# B&R Automation Studio project TD52 (part 68)

#### Gen2_ref.h
```c
/********************************************************************
 * COPYRIGHT -- B&R Industrial Automation GmbH
 ********************************************************************
 * Program: Gen2_ref
 * File: Gen2_ref.h
 * Author: 105055527
 * Last modified by: kelleto00
 * Created: Wed Apr 16 13:02:53 2008
 * Last modified: Wed Oct 09 10:01:33 2024
 * Model Version: 4.14.00.04
 * Description: V4.10.00.01, 01-09-2020 Keller, Ke Estimator, additive LS factor, Ptraj SpeedCtrl, LVRT Freeze HLCi
   V4.10.00.01, 02-10-2020 Keller, bugfix HLCi p2srefLX init, BDC_lib: change Inf to 1e7
   V4.10.00.01, 13-11-2020 Keller, bugfix LXcorr T2s/ZZP, LSLff damping, dbgOut for Leanox WG compensation
   V4.10.00.01, 27-01-2021 Keller, Lx WGV compensation: no reset in island mode, addition before skipfire compensation
   V4.10.00.01, 02-02-2021 Keller, initialization lambda estimation with rLam_Start
   V4.11.00.01, 28-05-2021 Keller, Gas Quality Change (GQC) Improvements, LHV estimator output
   V4.11.00.01, 05-11-2021 Keller, Bugfix BDC: worksplit offset, optionally Nset instead of Nnom, rN_Eng_LRskipF
   V4.12.00.01, 10-02-2021 Keller, SpeedCtrl2.0 TU Wien: Disturbance Estimator, LQR incl. droop & leanox
   V4.12.00.02, 23-05-2022 Arnold, Leanox point C in low load
   V4.12.00.02, 09-06-2022 Kafka, add external skip fire input for isolated and grid parallel operation
   V4.12.00.03, 15-09-2022 Keller, add power trajectory to HLCi for extended LQR (Droop setpoint)
   V4.12.00.04, 12-10-2022 Keller, add gas flow comp. factor for rejections
   V4.12.00.05, 13-10-2022 Keller, power filter for static skipfire in island mode
   V4.12.00.06, 15-11-2022 Keller, Ke adaptation with disturbance observer
   V4.13.00.01, 15-11-2022 Keller, FDC: R_mix output, HLCi: R_mix for Ke
   V4.13.00.02, 10-07-2023 Keller, interpolation of LHV, rho_gas and Lmin
   V4.13.00.03, 10-07-2023 Keller, load dependent gas dosage delay
   V4.13.00.04, 11-09-2023 Keller, D-part FSM, bugfix dPTV ramp
   V4.13.00.05, 27-02-2024 Keller, Filter outputs without bSS
   V4.13.00.06, 10-04-2024 Keller, bugfix leanox manual mode with bSepEmisCtrl
   V4.14.00.01, 01-07-2024 Keller, iNskip_LRfor Ke calculation
   V4.14.00.02, 17-09-2024 Keller, Use actual speed for observer disturbance dg (Gen2_ref/HLC_Island (HLC_Island_ref)/iLQR_SF/Ref LQR)
   V4.14.00.03, 30-09-2024 Keller, LR gas flow compensation possible without actuator saturation
   V4.14.00.04, 02-10-2024 Keller, Limit derivative power setpoint for FSM
 * modified Comment:
 ********************************************************************
 * Header for program Gen2_ref
 ********************************************************************
 * Generated with B&R Automation Studio Target for Simulink V6.7.1
 * (ERT based)
 ********************************************************************/

#ifndef RTW_HEADER_Gen2_ref_h_
#define RTW_HEADER_Gen2_ref_h_
#include <math.h>
#ifndef Gen2_ref_COMMON_INCLUDES_
#define Gen2_ref_COMMON_INCLUDES_
#include "rtwtypes.h"
#include "zero_crossing_types.h"
#endif                                 /* Gen2_ref_COMMON_INCLUDES_ */

#include "Gen2_ref_types.h"
#include "lGen2.h"
/* Beginning of Dynamic TypeDefs: */
/* End of Dynamic TypeDefs: */
#ifndef MIN
#define MIN(a,b)	((a) < (b) ? (a) : (b))
#endif

#ifndef MAX
#define MAX(a,b)	((a) > (b) ? (a) : (b))
#endif

#ifndef AST_ROUND
#define AST_ROUND(x) ((x)>=0?(long long)((x)+0.5):(long long)((x)-0.5))
#endif

#include "rt_nonfinite.h"
#include "rt_defines.h"

/* Macros for accessing real-time model data structure */
#ifndef rtmGetBlockIO
#define rtmGetBlockIO(rtm)             ((rtm)->blockIO)
#endif

#ifndef rtmSetBlockIO
#define rtmSetBlockIO(rtm, val)        ((rtm)->blockIO = (val))
#endif

#ifndef rtmGetPrevZCSigState
#define rtmGetPrevZCSigState(rtm)      ((rtm)->prevZCSigState)
#endif

#ifndef rtmSetPrevZCSigState
#define rtmSetPrevZCSigState(rtm, val) ((rtm)->prevZCSigState = (val))
#endif

#ifndef rtmGetRootDWork
#define rtmGetRootDWork(rtm)           ((rtm)->dwork)
#endif

#ifndef rtmSetRootDWork
#define rtmSetRootDWork(rtm, val)      ((rtm)->dwork = (val))
#endif

#ifndef rtmGetY
#define rtmGetY(rtm)                   ((rtm)->outputs)
#endif

#ifndef rtmSetY
#define rtmSetY(rtm, val)              ((rtm)->outputs = (val))
#endif

#ifndef rtmGetErrorStatus
#define rtmGetErrorStatus(rtm)         ((rtm)->errorStatus)
#endif

#ifndef rtmSetErrorStatus
#define rtmSetErrorStatus(rtm, val)    ((rtm)->errorStatus = (val))
#endif

#ifndef MIN
#define MIN(a,b)                       ((a) < (b) ? (a) : (b))
#endif

#ifndef MAX
#define MAX(a,b)                       ((a) > (b) ? (a) : (b))
#endif

#ifndef AST_ROUND
#define AST_ROUND(x)                   ((x)>=0?(long long)((x)+0.5):(long long)((x)-0.5))
#endif

/* Block signals for system '<S23>/Filter1' */

/* Block states (default storage) for system '<S23>/Filter1' */

/* Block signals for system '<S23>/TON_1' */

/* Block states (default storage) for system '<S23>/TON_1' */

/* Block signals for system '<S62>/Filter3' */

/* Block states (default storage) for system '<S62>/Filter3' */

/* Block signals for system '<S24>/MATLAB Function' */

/* Block states (default storage) for system '<S24>/MATLAB Function' */

/* Block signals for system '<S27>/engine massflow' */

/* Block signals for system '<S1>/IntegerZOH' */

/* Block states (default storage) for system '<S1>/IntegerZOH' */

/* Block signals for system '<S144>/lam2cg1' */

/* Block signals for system '<S44>/engine massflow2' */

/* Block signals for system '<S161>/Inverse_Linearization4' */

/* Block signals for system '<S190>/N_TC_HP_filt' */

/* Block states (default storage) for system '<S190>/N_TC_HP_filt' */

/* Block signals for system '<S267>/Mg' */

/* Block signals for system '<S267>/lam2cg1' */

/* Block signals for system '<S305>/FILTER no delay' */

/* Block states (default storage) for system '<S305>/FILTER no delay' */

/* Block signals for system '<S306>/2nd Order Filter' */

/* Block states (default storage) for system '<S306>/2nd Order Filter' */

/* Block signals for system '<S306>/2nd Order Filter3' */

/* Block states (default storage) for system '<S306>/2nd Order Filter3' */

/* Block signals for system '<S6>/TOF' */

/* Block states (default storage) for system '<S6>/TOF' */

/* Block signals for system '<S373>/2-point interpolation, with extrapolation' */

/* Block signals for system '<S379>/MATLAB Function' */

/* Block states (default storage) for system '<S379>/MATLAB Function' */

/* Block signals for system '<S379>/MATLAB Function1' */

/* Block states (default storage) for system '<S379>/MATLAB Function1' */

/* Block signals for system '<S344>/Pd_filt' */

/* Block states (default storage) for system '<S344>/Pd_filt' */

/* Block signals for system '<S426>/TP' */

/* Block states (default storage) for system '<S426>/TP' */

/* Block signals for system '<S427>/TOF' */

/* Block states (default storage) for system '<S427>/TOF' */

/* Block signals for system '<S427>/TP_ActSat_CBV' */

/* Block states (default storage) for system '<S427>/TP_ActSat_CBV' */

/* Block signals for system '<S589>/MATLAB Function' */

/* Block states (default storage) for system '<S589>/MATLAB Function' */

/* Block signals for system '<S630>/Filter' */

/* Block states (default storage) for system '<S630>/Filter' */

/* Block signals for system '<S666>/Ke Map Update' */

/* Block states (default storage) for system '<S666>/Ke Map Update' */

/* Block signals for system '<S666>/MATLAB Function1' */

/* Block states (default storage) for system '<S666>/MATLAB Function1' */

/* Block signals (default storage) */

/* Block states (default storage) for system '<Root>' */

/* Zero-crossing (trigger) state */

/* Invariant block signals for system '<S306>/2nd Order Filter' */

/* Invariant block signals for system '<S306>/2nd Order Filter3' */

/* Invariant block signals for system '<S630>/Filter' */

/* Invariant block signals for system '<S666>/Ke Map Update' */

/* Invariant block signals (default storage) */

/* Constant parameters (default storage) */

/* External outputs (root outports fed by signals with default storage) */

/* Real-time Model Data Structure */

extern const ConstBlockIO_Gen2_ref Gen2_ref_ConstB;/* constant block i/o */

/* Constant parameters (default storage) */
extern const ConstParam_Gen2_ref Gen2_ref_ConstP;

/* Model entry point functions */
extern void Gen2_ref_initialize(RT_MODEL_Gen2_ref *const Gen2_ref_M, struct Gen2* inst);
extern void Gen2_ref_step(RT_MODEL_Gen2_ref *const Gen2_ref_M, struct Gen2* inst);
extern void Gen2_ref_terminate(RT_MODEL_Gen2_ref *const Gen2_ref_M, struct Gen2* inst);

/*-
 * The generated code includes comments that allow you to trace directly
 * back to the appropriate location in the model.  The basic format
 * is <system>/block_name, where system is the system number (uniquely
 * assigned by Simulink) and block_name is the name of the block.
 *
 * Use the MATLAB hilite_system command to trace the generated code back
 * to the model.  For example,
 *
 * hilite_system('<S3>')    - opens system 3
 * hilite_system('<S3>/Kp') - opens and selects block Kp which resides in S3
 *
 * Here is the system hierarchy for this model
 *
 * '<Root>' : 'Gen2_ref'
 * '<S1>'   : 'Gen2_ref/BDC'
 * '<S2>'   : 'Gen2_ref/DocBlock'
 * '<S3>'   : 'Gen2_ref/EFF'
 * '<S4>'   : 'Gen2_ref/EngineSignals'
 * '<S5>'   : 'Gen2_ref/FDC'
 * '<S6>'   : 'Gen2_ref/Gas Quality Change'
 * '<S7>'   : 'Gen2_ref/HLC_Grid'
 * '<S8>'   : 'Gen2_ref/HLC_Island'
 * '<S9>'   : 'Gen2_ref/ITC'
 * '<S10>'  : 'Gen2_ref/Info'
 * '<S11>'  : 'Gen2_ref/Interpolation gas 1//2&3 specific parameters'
 * '<S12>'  : 'Gen2_ref/Ke Estimator NetP'
 * '<S13>'  : 'Gen2_ref/LHV estimator'
 * '<S14>'  : 'Gen2_ref/LambdaLimit'
 * '<S15>'  : 'Gen2_ref/Leanox_Comp_WG'
 * '<S16>'  : 'Gen2_ref/Outputs'
 * '<S17>'  : 'Gen2_ref/Power trajectory'
 * '<S18>'  : 'Gen2_ref/Saturation Det'
 * '<S19>'  : 'Gen2_ref/Skipfire'
 * '<S20>'  : 'Gen2_ref/SteadyState'
 * '<S21>'  : 'Gen2_ref/brake eff estimate'
 * '<S22>'  : 'Gen2_ref/BDC/ TC Protection'
 * '<S23>'  : 'Gen2_ref/BDC/1_Motion_Planning3'
 * '<S24>'  : 'Gen2_ref/BDC/2_Approach_selector_TV'
 * '<S25>'  : 'Gen2_ref/BDC/Approach_selector_CBV'
 * '<S26>'  : 'Gen2_ref/BDC/CBV_Control'
 * '<S27>'  : 'Gen2_ref/BDC/CBV_Feedforward'
 * '<S28>'  : 'Gen2_ref/BDC/Compare To Constant'
 * '<S29>'  : 'Gen2_ref/BDC/Compare To Constant1'
 * '<S30>'  : 'Gen2_ref/BDC/Compare To Constant2'
 * '<S31>'  : 'Gen2_ref/BDC/Difference1'
 * '<S32>'  : 'Gen2_ref/BDC/Divisor'
 * '<S33>'  : 'Gen2_ref/BDC/Divisor1'
 * '<S34>'  : 'Gen2_ref/BDC/Divisor2'
 * '<S35>'  : 'Gen2_ref/BDC/Divisor3'
 * '<S36>'  : 'Gen2_ref/BDC/DocBlock'
 * '<S37>'  : 'Gen2_ref/BDC/IntegerZOH'
 * '<S38>'  : 'Gen2_ref/BDC/IntegerZOH1'
 * '<S39>'  : 'Gen2_ref/BDC/IntegerZOH2'
 * '<S40>'  : 'Gen2_ref/BDC/Model Info'
 * '<S41>'  : 'Gen2_ref/BDC/PID_para'
 * '<S42>'  : 'Gen2_ref/BDC/Saturation Dynamic'
 * '<S43>'  : 'Gen2_ref/BDC/SurgeProtection'
 * '<S44>'  : 'Gen2_ref/BDC/TV_Feedforward'
 * '<S45>'  : 'Gen2_ref/BDC/Throttle_Control'
 * '<S46>'  : 'Gen2_ref/BDC/WGV_Feedforward'
 * '<S47>'  : 'Gen2_ref/BDC/ TC Protection/Compare To Zero'
 * '<S48>'  : 'Gen2_ref/BDC/1_Motion_Planning3/Delta_ref'
 * '<S49>'  : 'Gen2_ref/BDC/1_Motion_Planning3/Filter1'
 * '<S50>'  : 'Gen2_ref/BDC/1_Motion_Planning3/Filter2'
 * '<S51>'  : 'Gen2_ref/BDC/1_Motion_Planning3/Filter4'
 * '<S52>'  : 'Gen2_ref/BDC/1_Motion_Planning3/Rate Limit'
 * '<S53>'  : 'Gen2_ref/BDC/1_Motion_Planning3/Reset_'
 * '<S54>'  : 'Gen2_ref/BDC/1_Motion_Planning3/Saturation Dynamic'
 * '<S55>'  : 'Gen2_ref/BDC/1_Motion_Planning3/Saturation Dynamic1'
 * '<S56>'  : 'Gen2_ref/BDC/1_Motion_Planning3/Saturation Dynamic2'
 * '<S57>'  : 'Gen2_ref/BDC/1_Motion_Planning3/Saturation Dynamic3'
 * '<S58>'  : 'Gen2_ref/BDC/1_Motion_Planning3/Saturation Dynamic4'
 * '<S59>'  : 'Gen2_ref/BDC/1_Motion_Planning3/Saturation Dynamic5'
 * '<S60>'  : 'Gen2_ref/BDC/1_Motion_Planning3/Saturation Dynamic6'
 * '<S61>'  : 'Gen2_ref/BDC/1_Motion_Planning3/TON_1'
 * '<S62>'  : 'Gen2_ref/BDC/1_Motion_Planning3/offset for LEANOX tracking if TV open'
 * '<S63>'  : 'Gen2_ref/BDC/1_Motion_Planning3/rateLimit'
 * '<S64>'  : 'Gen2_ref/BDC/1_Motion_Planning3/rateLimit1'
 * '<S65>'  : 'Gen2_ref/BDC/1_Motion_Planning3/ref traj'
 * '<S66>'  : 'Gen2_ref/BDC/1_Motion_Planning3/Delta_ref/Compare To Zero'
 * '<S67>'  : 'Gen2_ref/BDC/1_Motion_Planning3/Delta_ref/Divisor'
 * '<S68>'  : 'Gen2_ref/BDC/1_Motion_Planning3/Delta_ref/Divisor1'
 * '<S69>'  : 'Gen2_ref/BDC/1_Motion_Planning3/Delta_ref/Divisor/Data Type Conversion Inherited'
 * '<S70>'  : 'Gen2_ref/BDC/1_Motion_Planning3/Delta_ref/Divisor1/Data Type Conversion Inherited'
 * '<S71>'  : 'Gen2_ref/BDC/1_Motion_Planning3/Filter1/Divisor'
 * '<S72>'  : 'Gen2_ref/BDC/1_Motion_Planning3/Filter1/Divisor/Data Type Conversion Inherited'
 * '<S73>'  : 'Gen2_ref/BDC/1_Motion_Planning3/Filter2/Divisor'
 * '<S74>'  : 'Gen2_ref/BDC/1_Motion_Planning3/Filter2/Divisor/Data Type Conversion Inherited'
 * '<S75>'  : 'Gen2_ref/BDC/1_Motion_Planning3/Filter4/Divisor'
 * '<S76>'  : 'Gen2_ref/BDC/1_Motion_Planning3/Filter4/Divisor/Data Type Conversion Inherited'
 * '<S77>'  : 'Gen2_ref/BDC/1_Motion_Planning3/Rate Limit/slewratelimit_rejection CBV'
 * '<S78>'  : 'Gen2_ref/BDC/1_Motion_Planning3/Rate Limit/slewratelimit_rejection TV'
 * '<S79>'  : 'Gen2_ref/BDC/1_Motion_Planning3/Rate Limit/slewratelimit_rejection CBV/rateLimit'
 * '<S80>'  : 'Gen2_ref/BDC/1_Motion_Planning3/Rate Limit/slewratelimit_rejection CBV/rateLimit1'
 * '<S81>'  : 'Gen2_ref/BDC/1_Motion_Planning3/Rate Limit/slewratelimit_rejection CBV/rateLimit2'
 * '<S82>'  : 'Gen2_ref/BDC/1_Motion_Planning3/Rate Limit/slewratelimit_rejection CBV/rateLimit3'
 * '<S83>'  : 'Gen2_ref/BDC/1_Motion_Planning3/Rate Limit/slewratelimit_rejection CBV/rateLimit/Saturation Dynamic'
 * '<S84>'  : 'Gen2_ref/BDC/1_Motion_Planning3/Rate Limit/slewratelimit_rejection CBV/rateLimit1/Saturation Dynamic'
 * '<S85>'  : 'Gen2_ref/BDC/1_Motion_Planning3/Rate Limit/slewratelimit_rejection CBV/rateLimit2/Saturation Dynamic'
 * '<S86>'  : 'Gen2_ref/BDC/1_Motion_Planning3/Rate Limit/slewratelimit_rejection CBV/rateLimit3/Saturation Dynamic'
 * '<S87>'  : 'Gen2_ref/BDC/1_Motion_Planning3/Rate Limit/slewratelimit_rejection TV/rateLimit'
 * '<S88>'  : 'Gen2_ref/BDC/1_Motion_Planning3/Rate Limit/slewratelimit_rejection TV/rateLimit1'
 * '<S89>'  : 'Gen2_ref/BDC/1_Motion_Planning3/Rate Limit/slewratelimit_rejection TV/rateLimit2'
 * '<S90>'  : 'Gen2_ref/BDC/1_Motion_Planning3/Rate Limit/slewratelimit_rejection TV/rateLimit3'
 * '<S91>'  : 'Gen2_ref/BDC/1_Motion_Planning3/Rate Limit/slewratelimit_rejection TV/rateLimit/Saturation Dynamic'
 * '<S92>'  : 'Gen2_ref/BDC/1_Motion_Planning3/Rate Limit/slewratelimit_rejection TV/rateLimit1/Saturation Dynamic'
 * '<S93>'  : 'Gen2_ref/BDC/1_Motion_Planning3/Rate Limit/slewratelimit_rejection TV/rateLimit2/Saturation Dynamic'
 * '<S94>'  : 'Gen2_ref/BDC/1_Motion_Planning3/Rate Limit/slewratelimit_rejection TV/rateLimit3/Saturation Dynamic'
 * '<S95>'  : 'Gen2_ref/BDC/1_Motion_Planning3/TON_1/Data Type Conversion Inherited'
 * '<S96>'  : 'Gen2_ref/BDC/1_Motion_Planning3/offset for LEANOX tracking if TV open/Divisor'
 * '<S97>'  : 'Gen2_ref/BDC/1_Motion_Planning3/offset for LEANOX tracking if TV open/Filter3'
 * '<S98>'  : 'Gen2_ref/BDC/1_Motion_Planning3/offset for LEANOX tracking if TV open/MATLAB Function'
 * '<S99>'  : 'Gen2_ref/BDC/1_Motion_Planning3/offset for LEANOX tracking if TV open/Divisor/Data Type Conversion Inherited'
 * '<S100>' : 'Gen2_ref/BDC/1_Motion_Planning3/offset for LEANOX tracking if TV open/Filter3/Divisor'
 * '<S101>' : 'Gen2_ref/BDC/1_Motion_Planning3/offset for LEANOX tracking if TV open/Filter3/Divisor/Data Type Conversion Inherited'
 * '<S102>' : 'Gen2_ref/BDC/1_Motion_Planning3/rateLimit/Saturation Dynamic'
 * '<S103>' : 'Gen2_ref/BDC/1_Motion_Planning3/rateLimit1/Saturation Dynamic'
 * '<S104>' : 'Gen2_ref/BDC/2_Approach_selector_TV/MATLAB Function'
 * '<S105>' : 'Gen2_ref/BDC/Approach_selector_CBV/MATLAB Function'
 * '<S106>' : 'Gen2_ref/BDC/Approach_selector_CBV/Saturation Dynamic'
 * '<S107>' : 'Gen2_ref/BDC/CBV_Control/Detect Change'
 * '<S108>' : 'Gen2_ref/BDC/CBV_Control/Saturation Dynamic'
 * '<S109>' : 'Gen2_ref/BDC/CBV_Control/Saturation Dynamic1'
 * '<S110>' : 'Gen2_ref/BDC/CBV_Control/fb_err'
 * '<S111>' : 'Gen2_ref/BDC/CBV_Control/reset init'
 * '<S112>' : 'Gen2_ref/BDC/CBV_Feedforward/Divisor'
 * '<S113>' : 'Gen2_ref/BDC/CBV_Feedforward/MATLAB Function1'
 * '<S114>' : 'Gen2_ref/BDC/CBV_Feedforward/Saturation Dynamic'
 * '<S115>' : 'Gen2_ref/BDC/CBV_Feedforward/Saturation Dynamic1'
 * '<S116>' : 'Gen2_ref/BDC/CBV_Feedforward/cbv tracking1'
 * '<S117>' : 'Gen2_ref/BDC/CBV_Feedforward/dynamic_massflow '
 * '<S118>' : 'Gen2_ref/BDC/CBV_Feedforward/engine massflow'
 * '<S119>' : 'Gen2_ref/BDC/CBV_Feedforward/engine massflow1'
 * '<S120>' : 'Gen2_ref/BDC/CBV_Feedforward/Divisor/Data Type Conversion Inherited'
 * '<S121>' : 'Gen2_ref/BDC/CBV_Feedforward/cbv tracking1/Compare To Constant'
 * '<S122>' : 'Gen2_ref/BDC/CBV_Feedforward/cbv tracking1/Compare To Constant1'
 * '<S123>' : 'Gen2_ref/BDC/CBV_Feedforward/cbv tracking1/Saturation Dynamic'
 * '<S124>' : 'Gen2_ref/BDC/Divisor/Data Type Conversion Inherited'
 * '<S125>' : 'Gen2_ref/BDC/Divisor1/Data Type Conversion Inherited'
 * '<S126>' : 'Gen2_ref/BDC/Divisor2/Data Type Conversion Inherited'
 * '<S127>' : 'Gen2_ref/BDC/Divisor3/Data Type Conversion Inherited'
 * '<S128>' : 'Gen2_ref/BDC/PID_para/Saturation Dynamic'
 * '<S129>' : 'Gen2_ref/BDC/PID_para/Saturation Dynamic1'
 * '<S130>' : 'Gen2_ref/BDC/PID_para/Saturation Dynamic2'
 * '<S131>' : 'Gen2_ref/BDC/PID_para/Saturation Dynamic3'
 * '<S132>' : 'Gen2_ref/BDC/PID_para/p2s fitler2'
 * '<S133>' : 'Gen2_ref/BDC/SurgeProtection/SP'
 * '<S134>' : 'Gen2_ref/BDC/SurgeProtection/SP2'
 * '<S135>' : 'Gen2_ref/BDC/SurgeProtection/SP/Divisor'
 * '<S136>' : 'Gen2_ref/BDC/SurgeProtection/SP/Saturation Dynamic'
 * '<S137>' : 'Gen2_ref/BDC/SurgeProtection/SP/Saturation Dynamic1'
 * '<S138>' : 'Gen2_ref/BDC/SurgeProtection/SP/Divisor/Data Type Conversion Inherited'
 * '<S139>' : 'Gen2_ref/BDC/SurgeProtection/SP2/Divisor'
 * '<S140>' : 'Gen2_ref/BDC/SurgeProtection/SP2/Divisor2'
 * '<S141>' : 'Gen2_ref/BDC/SurgeProtection/SP2/Filter'
 * '<S142>' : 'Gen2_ref/BDC/SurgeProtection/SP2/MATLAB Function'
 * '<S143>' : 'Gen2_ref/BDC/SurgeProtection/SP2/MATLAB Function1'
 * '<S144>' : 'Gen2_ref/BDC/SurgeProtection/SP2/MassFlowCalc'
 * '<S145>' : 'Gen2_ref/BDC/SurgeProtection/SP2/Divisor/Data Type Conversion Inherited'
 * '<S146>' : 'Gen2_ref/BDC/SurgeProtection/SP2/Divisor2/Data Type Conversion Inherited'
 * '<S147>' : 'Gen2_ref/BDC/SurgeProtection/SP2/Filter/Divisor'
 * '<S148>' : 'Gen2_ref/BDC/SurgeProtection/SP2/Filter/Divisor/Data Type Conversion Inherited'
 * '<S149>' : 'Gen2_ref/BDC/SurgeProtection/SP2/MassFlowCalc/Divisor2'
 * '<S150>' : 'Gen2_ref/BDC/SurgeProtection/SP2/MassFlowCalc/lam2cg1'
 * '<S151>' : 'Gen2_ref/BDC/SurgeProtection/SP2/MassFlowCalc/Divisor2/Data Type Conversion Inherited'
 * '<S152>' : 'Gen2_ref/BDC/SurgeProtection/SP2/MassFlowCalc/lam2cg1/Divisor'
 * '<S153>' : 'Gen2_ref/BDC/SurgeProtection/SP2/MassFlowCalc/lam2cg1/Divisor/Data Type Conversion Inherited'
 * '<S154>' : 'Gen2_ref/BDC/TV_Feedforward/Divisor'
 * '<S155>' : 'Gen2_ref/BDC/TV_Feedforward/Dyn_Term'
 * '<S156>' : 'Gen2_ref/BDC/TV_Feedforward/MATLAB Function3'
 * '<S157>' : 'Gen2_ref/BDC/TV_Feedforward/Saturation Dynamic1'
 * '<S158>' : 'Gen2_ref/BDC/TV_Feedforward/engine massflow2'
 * '<S159>' : 'Gen2_ref/BDC/TV_Feedforward/Divisor/Data Type Conversion Inherited'
 * '<S160>' : 'Gen2_ref/BDC/Throttle_Control/Detect Change'
 * '<S161>' : 'Gen2_ref/BDC/Throttle_Control/Integrator Init'
 * '<S162>' : 'Gen2_ref/BDC/Throttle_Control/Inverse_Linearization1'
 * '<S163>' : 'Gen2_ref/BDC/Throttle_Control/Inverse_Linearization2'
 * '<S164>' : 'Gen2_ref/BDC/Throttle_Control/Inverse_Linearization3'
 * '<S165>' : 'Gen2_ref/BDC/Throttle_Control/Inverse_Linearization4'
 * '<S166>' : 'Gen2_ref/BDC/Throttle_Control/Linearization'
 * '<S167>' : 'Gen2_ref/BDC/Throttle_Control/Saturation Dynamic'
 * '<S168>' : 'Gen2_ref/BDC/Throttle_Control/tv_fb_err'
 * '<S169>' : 'Gen2_ref/BDC/Throttle_Control/Integrator Init/Inverse_Linearization4'
 * '<S170>' : 'Gen2_ref/BDC/WGV_Feedforward/Divisor'
 * '<S171>' : 'Gen2_ref/BDC/WGV_Feedforward/MATLAB Function1'
 * '<S172>' : 'Gen2_ref/BDC/WGV_Feedforward/Saturation Dynamic'
 * '<S173>' : 'Gen2_ref/BDC/WGV_Feedforward/Saturation Dynamic1'
 * '<S174>' : 'Gen2_ref/BDC/WGV_Feedforward/cbv tracking1'
 * '<S175>' : 'Gen2_ref/BDC/WGV_Feedforward/dynamic_massflow'
 * '<S176>' : 'Gen2_ref/BDC/WGV_Feedforward/engine massflow'
 * '<S177>' : 'Gen2_ref/BDC/WGV_Feedforward/engine massflow1'
 * '<S178>' : 'Gen2_ref/BDC/WGV_Feedforward/Divisor/Data Type Conversion Inherited'
 * '<S179>' : 'Gen2_ref/BDC/WGV_Feedforward/cbv tracking1/Compare To Constant'
 * '<S180>' : 'Gen2_ref/BDC/WGV_Feedforward/cbv tracking1/Saturation Dynamic'
 * '<S181>' : 'Gen2_ref/BDC/WGV_Feedforward/cbv tracking1/TP'
 * '<S182>' : 'Gen2_ref/BDC/WGV_Feedforward/cbv tracking1/TP/Compare To Zero'
 * '<S183>' : 'Gen2_ref/BDC/WGV_Feedforward/cbv tracking1/TP/Enabled Subsystem'
 * '<S184>' : 'Gen2_ref/BDC/WGV_Feedforward/cbv tracking1/TP/Enabled Subsystem1'
 * '<S185>' : 'Gen2_ref/BDC/WGV_Feedforward/cbv tracking1/TP/Rate Limiter'
 * '<S186>' : 'Gen2_ref/BDC/WGV_Feedforward/cbv tracking1/TP/Rate Limiter/Saturation Dynamic'
 * '<S187>' : 'Gen2_ref/EngineSignals/Compare To Constant'
 * '<S188>' : 'Gen2_ref/EngineSignals/Compare To Constant1'
 * '<S189>' : 'Gen2_ref/EngineSignals/Compare To Constant3'
 * '<S190>' : 'Gen2_ref/EngineSignals/IgnAvg'
 * '<S191>' : 'Gen2_ref/EngineSignals/N_TC_HP_filt'
 * '<S192>' : 'Gen2_ref/EngineSignals/N_TC_LP_filt'
 * '<S193>' : 'Gen2_ref/EngineSignals/N_TC_LP_filt1'
 * '<S194>' : 'Gen2_ref/EngineSignals/Pel_filt'
 * '<S195>' : 'Gen2_ref/EngineSignals/T1HP_filt'
 * '<S196>' : 'Gen2_ref/EngineSignals/T1LP_filt'
 * '<S197>' : 'Gen2_ref/EngineSignals/T2s_filt'
 * '<S198>' : 'Gen2_ref/EngineSignals/T3HP_filt'
 * '<S199>' : 'Gen2_ref/EngineSignals/T3LP_filt'
 * '<S200>' : 'Gen2_ref/EngineSignals/T4LP_filt'
 * '<S201>' : 'Gen2_ref/EngineSignals/Volt_filt'
 * '<S202>' : 'Gen2_ref/EngineSignals/p1HP_filt'
 * '<S203>' : 'Gen2_ref/EngineSignals/p1LP_filt'
 * '<S204>' : 'Gen2_ref/EngineSignals/p2HP_filt'
 * '<S205>' : 'Gen2_ref/EngineSignals/p2s_filt'
 * '<S206>' : 'Gen2_ref/EngineSignals/p3LP_filt'
 * '<S207>' : 'Gen2_ref/EngineSignals/p3LP_filt1'
 * '<S208>' : 'Gen2_ref/EngineSignals/p4LP_filt'
 * '<S209>' : 'Gen2_ref/EngineSignals/IgnAvg/N_TC_HP_filt'
 * '<S210>' : 'Gen2_ref/EngineSignals/IgnAvg/N_TC_HP_filt/Divisor'
 * '<S211>' : 'Gen2_ref/EngineSignals/IgnAvg/N_TC_HP_filt/Divisor/Data Type Conversion Inherited'
 * '<S212>' : 'Gen2_ref/EngineSignals/N_TC_HP_filt/N_TC_HP_filt'
 * '<S213>' : 'Gen2_ref/EngineSignals/N_TC_HP_filt/N_TC_HP_filt/Divisor'
 * '<S214>' : 'Gen2_ref/EngineSignals/N_TC_HP_filt/N_TC_HP_filt/Divisor/Data Type Conversion Inherited'
 * '<S215>' : 'Gen2_ref/EngineSignals/N_TC_LP_filt/N_TC_LP_filt'
 * '<S216>' : 'Gen2_ref/EngineSignals/N_TC_LP_filt/N_TC_LP_filt/Divisor'
 * '<S217>' : 'Gen2_ref/EngineSignals/N_TC_LP_filt/N_TC_LP_filt/Divisor/Data Type Conversion Inherited'
 * '<S218>' : 'Gen2_ref/EngineSignals/N_TC_LP_filt1/N_TC_LP_filt'
 * '<S219>' : 'Gen2_ref/EngineSignals/N_TC_LP_filt1/N_TC_LP_filt/Divisor'
 * '<S220>' : 'Gen2_ref/EngineSignals/N_TC_LP_filt1/N_TC_LP_filt/Divisor/Data Type Conversion Inherited'
 * '<S221>' : 'Gen2_ref/EngineSignals/Pel_filt/Pel_filt'
 * '<S222>' : 'Gen2_ref/EngineSignals/Pel_filt/Pel_filt/Divisor'
 * '<S223>' : 'Gen2_ref/EngineSignals/Pel_filt/Pel_filt/Divisor/Data Type Conversion Inherited'
 * '<S224>' : 'Gen2_ref/EngineSignals/T1HP_filt/T1HP_filt'
 * '<S225>' : 'Gen2_ref/EngineSignals/T1HP_filt/T1HP_filt/Divisor'
 * '<S226>' : 'Gen2_ref/EngineSignals/T1HP_filt/T1HP_filt/Divisor/Data Type Conversion Inherited'
 * '<S227>' : 'Gen2_ref/EngineSignals/T1LP_filt/T1LP_filt'
 * '<S228>' : 'Gen2_ref/EngineSignals/T1LP_filt/T1LP_filt/Divisor'
 * '<S229>' : 'Gen2_ref/EngineSignals/T1LP_filt/T1LP_filt/Divisor/Data Type Conversion Inherited'
 * '<S230>' : 'Gen2_ref/EngineSignals/T2s_filt/T2s_filt'
 * '<S231>' : 'Gen2_ref/EngineSignals/T2s_filt/T2s_filt/Divisor'
 * '<S232>' : 'Gen2_ref/EngineSignals/T2s_filt/T2s_filt/Divisor/Data Type Conversion Inherited'
 * '<S233>' : 'Gen2_ref/EngineSignals/T3HP_filt/T3HP_filt'
 * '<S234>' : 'Gen2_ref/EngineSignals/T3HP_filt/T3HP_filt/Divisor'
 * '<S235>' : 'Gen2_ref/EngineSignals/T3HP_filt/T3HP_filt/Divisor/Data Type Conversion Inherited'
 * '<S236>' : 'Gen2_ref/EngineSignals/T3LP_filt/T3LP_filt'
 * '<S237>' : 'Gen2_ref/EngineSignals/T3LP_filt/T3LP_filt/Divisor'
 * '<S238>' : 'Gen2_ref/EngineSignals/T3LP_filt/T3LP_filt/Divisor/Data Type Conversion Inherited'
 * '<S239>' : 'Gen2_ref/EngineSignals/T4LP_filt/T3LP_filt'
 * '<S240>' : 'Gen2_ref/EngineSignals/T4LP_filt/T3LP_filt/Divisor'
 * '<S241>' : 'Gen2_ref/EngineSignals/T4LP_filt/T3LP_filt/Divisor/Data Type Conversion Inherited'
 * '<S242>' : 'Gen2_ref/EngineSignals/Volt_filt/Volt_filt'
 * '<S243>' : 'Gen2_ref/EngineSignals/Volt_filt/Volt_filt/Divisor'
 * '<S244>' : 'Gen2_ref/EngineSignals/Volt_filt/Volt_filt/Divisor/Data Type Conversion Inherited'
 * '<S245>' : 'Gen2_ref/EngineSignals/p1HP_filt/p1HP_filt'
 * '<S246>' : 'Gen2_ref/EngineSignals/p1HP_filt/p1HP_filt/Divisor'
 * '<S247>' : 'Gen2_ref/EngineSignals/p1HP_filt/p1HP_filt/Divisor/Data Type Conversion Inherited'
 * '<S248>' : 'Gen2_ref/EngineSignals/p1LP_filt/Filter'
 * '<S249>' : 'Gen2_ref/EngineSignals/p1LP_filt/Filter/Divisor'
 * '<S250>' : 'Gen2_ref/EngineSignals/p1LP_filt/Filter/Divisor/Data Type Conversion Inherited'
 * '<S251>' : 'Gen2_ref/EngineSignals/p2HP_filt/p2HP_filt'
 * '<S252>' : 'Gen2_ref/EngineSignals/p2HP_filt/p2HP_filt/Divisor'
 * '<S253>' : 'Gen2_ref/EngineSignals/p2HP_filt/p2HP_filt/Divisor/Data Type Conversion Inherited'
 * '<S254>' : 'Gen2_ref/EngineSignals/p2s_filt/p2s_filt'
 * '<S255>' : 'Gen2_ref/EngineSignals/p2s_filt/p2s_filt/Divisor'
 * '<S256>' : 'Gen2_ref/EngineSignals/p2s_filt/p2s_filt/Divisor/Data Type Conversion Inherited'
 * '<S257>' : 'Gen2_ref/EngineSignals/p3LP_filt/p3LP_filt'
 * '<S258>' : 'Gen2_ref/EngineSignals/p3LP_filt/p3LP_filt/Divisor'
 * '<S259>' : 'Gen2_ref/EngineSignals/p3LP_filt/p3LP_filt/Divisor/Data Type Conversion Inherited'
 * '<S260>' : 'Gen2_ref/EngineSignals/p3LP_filt1/p3LP_filt'
 * '<S261>' : 'Gen2_ref/EngineSignals/p3LP_filt1/p3LP_filt/Divisor'
 * '<S262>' : 'Gen2_ref/EngineSignals/p3LP_filt1/p3LP_filt/Divisor/Data Type Conversion Inherited'
 * '<S263>' : 'Gen2_ref/EngineSignals/p4LP_filt/p4LP_filt'
 * '<S264>' : 'Gen2_ref/EngineSignals/p4LP_filt/p4LP_filt/Divisor'
 * '<S265>' : 'Gen2_ref/EngineSignals/p4LP_filt/p4LP_filt/Divisor/Data Type Conversion Inherited'
 * '<S266>' : 'Gen2_ref/FDC/DocBlock'
 * '<S267>' : 'Gen2_ref/FDC/GasArt12'
 * '<S268>' : 'Gen2_ref/FDC/GasArt3'
 * '<S269>' : 'Gen2_ref/FDC/IntegerZOH'
 * '<S270>' : 'Gen2_ref/FDC/IntegerZOH1'
 * '<S271>' : 'Gen2_ref/FDC/Model Info'
 * '<S272>' : 'Gen2_ref/FDC/Signal Conditioning'
 * '<S273>' : 'Gen2_ref/FDC/GasArt12/Divisor'
 * '<S274>' : 'Gen2_ref/FDC/GasArt12/Mg'
 * '<S275>' : 'Gen2_ref/FDC/GasArt12/Safety check logic'
 * '<S276>' : 'Gen2_ref/FDC/GasArt12/lam2cg'
 * '<S277>' : 'Gen2_ref/FDC/GasArt12/lam2cg1'
 * '<S278>' : 'Gen2_ref/FDC/GasArt12/Divisor/Data Type Conversion Inherited'
 * '<S279>' : 'Gen2_ref/FDC/GasArt12/Mg/Divisor'
 * '<S280>' : 'Gen2_ref/FDC/GasArt12/Mg/Divisor/Data Type Conversion Inherited'
 * '<S281>' : 'Gen2_ref/FDC/GasArt12/Safety check logic/Divisor1'
 * '<S282>' : 'Gen2_ref/FDC/GasArt12/Safety check logic/Divisor2'
 * '<S283>' : 'Gen2_ref/FDC/GasArt12/Safety check logic/Divisor1/Data Type Conversion Inherited'
 * '<S284>' : 'Gen2_ref/FDC/GasArt12/Safety check logic/Divisor2/Data Type Conversion Inherited'
 * '<S285>' : 'Gen2_ref/FDC/GasArt12/lam2cg/Divisor'
 * '<S286>' : 'Gen2_ref/FDC/GasArt12/lam2cg/Divisor/Data Type Conversion Inherited'
 * '<S287>' : 'Gen2_ref/FDC/GasArt12/lam2cg1/Divisor'
 * '<S288>' : 'Gen2_ref/FDC/GasArt12/lam2cg1/Divisor/Data Type Conversion Inherited'
 * '<S289>' : 'Gen2_ref/FDC/GasArt3/Divisor'
 * '<S290>' : 'Gen2_ref/FDC/GasArt3/Mg'
 * '<S291>' : 'Gen2_ref/FDC/GasArt3/Safety check logic'
 * '<S292>' : 'Gen2_ref/FDC/GasArt3/lam2cg'
 * '<S293>' : 'Gen2_ref/FDC/GasArt3/lam2cg1'
 * '<S294>' : 'Gen2_ref/FDC/GasArt3/Divisor/Data Type Conversion Inherited'
 * '<S295>' : 'Gen2_ref/FDC/GasArt3/Mg/Divisor'
 * '<S296>' : 'Gen2_ref/FDC/GasArt3/Mg/Divisor/Data Type Conversion Inherited'
 * '<S297>' : 'Gen2_ref/FDC/GasArt3/Safety check logic/Divisor1'
 * '<S298>' : 'Gen2_ref/FDC/GasArt3/Safety check logic/Divisor2'
 * '<S299>' : 'Gen2_ref/FDC/GasArt3/Safety check logic/Divisor1/Data Type Conversion Inherited'
 * '<S300>' : 'Gen2_ref/FDC/GasArt3/Safety check logic/Divisor2/Data Type Conversion Inherited'
 * '<S301>' : 'Gen2_ref/FDC/GasArt3/lam2cg/Divisor'
 * '<S302>' : 'Gen2_ref/FDC/GasArt3/lam2cg/Divisor/Data Type Conversion Inherited'
 * '<S303>' : 'Gen2_ref/FDC/GasArt3/lam2cg1/Divisor'
 * '<S304>' : 'Gen2_ref/FDC/GasArt3/lam2cg1/Divisor/Data Type Conversion Inherited'
 * '<S305>' : 'Gen2_ref/FDC/Signal Conditioning/first order filter'
 * '<S306>' : 'Gen2_ref/FDC/Signal Conditioning/second order filter'
 * '<S307>' : 'Gen2_ref/FDC/Signal Conditioning/transient switching'
 * '<S308>' : 'Gen2_ref/FDC/Signal Conditioning/first order filter/FILTER no delay'
 * '<S309>' : 'Gen2_ref/FDC/Signal Conditioning/first order filter/FILTER no delay1'
 * '<S310>' : 'Gen2_ref/FDC/Signal Conditioning/first order filter/FILTER no delay2'
 * '<S311>' : 'Gen2_ref/FDC/Signal Conditioning/first order filter/FILTER no delay3'
 * '<S312>' : 'Gen2_ref/FDC/Signal Conditioning/first order filter/FILTER no delay4'
 * '<S313>' : 'Gen2_ref/FDC/Signal Conditioning/first order filter/FILTER no delay5'
 * '<S314>' : 'Gen2_ref/FDC/Signal Conditioning/second order filter/2nd Order Filter'
 * '<S315>' : 'Gen2_ref/FDC/Signal Conditioning/second order filter/2nd Order Filter1'
 * '<S316>' : 'Gen2_ref/FDC/Signal Conditioning/second order filter/2nd Order Filter2'
 * '<S317>' : 'Gen2_ref/FDC/Signal Conditioning/second order filter/2nd Order Filter3'
 * '<S318>' : 'Gen2_ref/FDC/Signal Conditioning/second order filter/2nd Order Filter4'
 * '<S319>' : 'Gen2_ref/FDC/Signal Conditioning/second order filter/2nd Order Filter/Divisor1'
 * '<S320>' : 'Gen2_ref/FDC/Signal Conditioning/second order filter/2nd Order Filter/Divisor1/Data Type Conversion Inherited'
 * '<S321>' : 'Gen2_ref/FDC/Signal Conditioning/second order filter/2nd Order Filter1/Divisor1'
 * '<S322>' : 'Gen2_ref/FDC/Signal Conditioning/second order filter/2nd Order Filter1/Divisor1/Data Type Conversion Inherited'
 * '<S323>' : 'Gen2_ref/FDC/Signal Conditioning/second order filter/2nd Order Filter2/Divisor1'
 * '<S324>' : 'Gen2_ref/FDC/Signal Conditioning/second order filter/2nd Order Filter2/Divisor1/Data Type Conversion Inherited'
 * '<S325>' : 'Gen2_ref/FDC/Signal Conditioning/second order filter/2nd Order Filter3/Divisor1'
 * '<S326>' : 'Gen2_ref/FDC/Signal Conditioning/second order filter/2nd Order Filter3/Divisor1/Data Type Conversion Inherited'
 * '<S327>' : 'Gen2_ref/FDC/Signal Conditioning/second order filter/2nd Order Filter4/Divisor1'
 * '<S328>' : 'Gen2_ref/FDC/Signal Conditioning/second order filter/2nd Order Filter4/Divisor1/Data Type Conversion Inherited'
 * '<S329>' : 'Gen2_ref/Gas Quality Change/TOF'
 * '<S330>' : 'Gen2_ref/Gas Quality Change/TOF1'
 * '<S331>' : 'Gen2_ref/Gas Quality Change/TOF2'
 * '<S332>' : 'Gen2_ref/Gas Quality Change/TON'
 * '<S333>' : 'Gen2_ref/Gas Quality Change/TOF/Data Type Conversion Inherited'
 * '<S334>' : 'Gen2_ref/Gas Quality Change/TOF1/Data Type Conversion Inherited'
 * '<S335>' : 'Gen2_ref/Gas Quality Change/TOF2/Data Type Conversion Inherited'
 * '<S336>' : 'Gen2_ref/Gas Quality Change/TON/Data Type Conversion Inherited'
 * '<S337>' : 'Gen2_ref/HLC_Grid/DocBlock'
 * '<S338>' : 'Gen2_ref/HLC_Grid/LEANOX map'
 * '<S339>' : 'Gen2_ref/HLC_Grid/LVRT_React'
 * '<S340>' : 'Gen2_ref/HLC_Grid/MBC_FF'
 * '<S341>' : 'Gen2_ref/HLC_Grid/Model Info'
 * '<S342>' : 'Gen2_ref/HLC_Grid/Power_Ctrl'
 * '<S343>' : 'Gen2_ref/HLC_Grid/Power_Ctrl Gas Quality Change'
 * '<S344>' : 'Gen2_ref/HLC_Grid/Power_Trajectory'
 * '<S345>' : 'Gen2_ref/HLC_Grid/Subsystem Reference'
 * '<S346>' : 'Gen2_ref/HLC_Grid/LEANOX map/Divisor'
 * '<S347>' : 'Gen2_ref/HLC_Grid/LEANOX map/Divisor1'
 * '<S348>' : 'Gen2_ref/HLC_Grid/LEANOX map/Divisor10'
 * '<S349>' : 'Gen2_ref/HLC_Grid/LEANOX map/Divisor11'
 * '<S350>' : 'Gen2_ref/HLC_Grid/LEANOX map/Divisor12'
 * '<S351>' : 'Gen2_ref/HLC_Grid/LEANOX map/Divisor2'
 * '<S352>' : 'Gen2_ref/HLC_Grid/LEANOX map/Divisor3'
 * '<S353>' : 'Gen2_ref/HLC_Grid/LEANOX map/Divisor4'
 * '<S354>' : 'Gen2_ref/HLC_Grid/LEANOX map/Divisor5'
 * '<S355>' : 'Gen2_ref/HLC_Grid/LEANOX map/Divisor6'
 * '<S356>' : 'Gen2_ref/HLC_Grid/LEANOX map/Divisor7'
 * '<S357>' : 'Gen2_ref/HLC_Grid/LEANOX map/Divisor8'
 * '<S358>' : 'Gen2_ref/HLC_Grid/LEANOX map/Divisor9'
 * '<S359>' : 'Gen2_ref/HLC_Grid/LEANOX map/LeanoxCorr'
 * '<S360>' : 'Gen2_ref/HLC_Grid/LEANOX map/Divisor/Data Type Conversion Inherited'
 * '<S361>' : 'Gen2_ref/HLC_Grid/LEANOX map/Divisor1/Data Type Conversion Inherited'
 * '<S362>' : 'Gen2_ref/HLC_Grid/LEANOX map/Divisor10/Data Type Conversion Inherited'
 * '<S363>' : 'Gen2_ref/HLC_Grid/LEANOX map/Divisor11/Data Type Conversion Inherited'
 * '<S364>' : 'Gen2_ref/HLC_Grid/LEANOX map/Divisor12/Data Type Conversion Inherited'
 * '<S365>' : 'Gen2_ref/HLC_Grid/LEANOX map/Divisor2/Data Type Conversion Inherited'
 * '<S366>' : 'Gen2_ref/HLC_Grid/LEANOX map/Divisor3/Data Type Conversion Inherited'
 * '<S367>' : 'Gen2_ref/HLC_Grid/LEANOX map/Divisor4/Data Type Conversion Inherited'
 * '<S368>' : 'Gen2_ref/HLC_Grid/LEANOX map/Divisor5/Data Type Conversion Inherited'
 * '<S369>' : 'Gen2_ref/HLC_Grid/LEANOX map/Divisor6/Data Type Conversion Inherited'
 * '<S370>' : 'Gen2_ref/HLC_Grid/LEANOX map/Divisor7/Data Type Conversion Inherited'
 * '<S371>' : 'Gen2_ref/HLC_Grid/LEANOX map/Divisor8/Data Type Conversion Inherited'
 * '<S372>' : 'Gen2_ref/HLC_Grid/LEANOX map/Divisor9/Data Type Conversion Inherited'
 * '<S373>' : 'Gen2_ref/HLC_Grid/LEANOX map/LeanoxCorr/Leanox_Comp'
 * '<S374>' : 'Gen2_ref/HLC_Grid/LEANOX map/LeanoxCorr/Leanox_Comp/2-point interpolation, with extrapolation'
 * '<S375>' : 'Gen2_ref/HLC_Grid/LEANOX map/LeanoxCorr/Leanox_Comp/2-point interpolation, with extrapolation1'
 * '<S376>' : 'Gen2_ref/HLC_Grid/LEANOX map/LeanoxCorr/Leanox_Comp/Saturation Dynamic'
 * '<S377>' : 'Gen2_ref/HLC_Grid/LEANOX map/LeanoxCorr/Leanox_Comp/Saturation Dynamic1'
 * '<S378>' : 'Gen2_ref/HLC_Grid/LVRT_React/MATLAB Function'
 * '<S379>' : 'Gen2_ref/HLC_Grid/Power_Ctrl/PID_Power'
 * '<S380>' : 'Gen2_ref/HLC_Grid/Power_Ctrl/Saturation Dynamic7'
 * '<S381>' : 'Gen2_ref/HLC_Grid/Power_Ctrl/Texh_limit'
 * '<S382>' : 'Gen2_ref/HLC_Grid/Power_Ctrl/PID_Power/MATLAB Function'
 * '<S383>' : 'Gen2_ref/HLC_Grid/Power_Ctrl/PID_Power/MATLAB Function1'
 * '<S384>' : 'Gen2_ref/HLC_Grid/Power_Ctrl/PID_Power/Saturation Dynamic'
 * '<S385>' : 'Gen2_ref/HLC_Grid/Power_Ctrl/PID_Power/rateLimit'
 * '<S386>' : 'Gen2_ref/HLC_Grid/Power_Ctrl/PID_Power/rateLimit/Saturation Dynamic'
 * '<S387>' : 'Gen2_ref/HLC_Grid/Power_Ctrl/Texh_limit/Saturation Dynamic4'
 * '<S388>' : 'Gen2_ref/HLC_Grid/Power_Ctrl Gas Quality Change/Anti Wind Up'
 * '<S389>' : 'Gen2_ref/HLC_Grid/Power_Ctrl Gas Quality Change/PID_Power'
 * '<S390>' : 'Gen2_ref/HLC_Grid/Power_Ctrl Gas Quality Change/Anti Wind Up/Saturation Dynamic'
 * '<S391>' : 'Gen2_ref/HLC_Grid/Power_Ctrl Gas Quality Change/PID_Power/MATLAB Function'
 * '<S392>' : 'Gen2_ref/HLC_Grid/Power_Ctrl Gas Quality Change/PID_Power/MATLAB Function1'
 * '<S393>' : 'Gen2_ref/HLC_Grid/Power_Ctrl Gas Quality Change/PID_Power/Saturation Dynamic'
 * '<S394>' : 'Gen2_ref/HLC_Grid/Power_Ctrl Gas Quality Change/PID_Power/rateLimit'
 * '<S395>' : 'Gen2_ref/HLC_Grid/Power_Ctrl Gas Quality Change/PID_Power/rateLimit/Saturation Dynamic'
 * '<S396>' : 'Gen2_ref/HLC_Grid/Power_Trajectory/Pd_filt'
 * '<S397>' : 'Gen2_ref/HLC_Grid/Power_Trajectory/Saturation Dynamic'
 * '<S398>' : 'Gen2_ref/HLC_Grid/Power_Trajectory/Saturation Dynamic1'
 * '<S399>' : 'Gen2_ref/HLC_Grid/Power_Trajectory/Saturation Dynamic2'
 * '<S400>' : 'Gen2_ref/HLC_Grid/Power_Trajectory/Saturation Dynamic3'
 * '<S401>' : 'Gen2_ref/HLC_Grid/Power_Trajectory/Saturation Dynamic4'
 * '<S402>' : 'Gen2_ref/HLC_Grid/Power_Trajectory/WO1'
 * '<S403>' : 'Gen2_ref/HLC_Grid/Power_Trajectory/WO2'
 * '<S404>' : 'Gen2_ref/HLC_Grid/Power_Trajectory/rateLimit'
 * '<S405>' : 'Gen2_ref/HLC_Grid/Power_Trajectory/Pd_filt/Divisor'
 * '<S406>' : 'Gen2_ref/HLC_Grid/Power_Trajectory/Pd_filt/Divisor/Data Type Conversion Inherited'
 * '<S407>' : 'Gen2_ref/HLC_Grid/Power_Trajectory/WO1/Divisor'
 * '<S408>' : 'Gen2_ref/HLC_Grid/Power_Trajectory/WO1/Divisor/Data Type Conversion Inherited'
 * '<S409>' : 'Gen2_ref/HLC_Grid/Power_Trajectory/WO2/Divisor'
 * '<S410>' : 'Gen2_ref/HLC_Grid/Power_Trajectory/WO2/Divisor/Data Type Conversion Inherited'
 * '<S411>' : 'Gen2_ref/HLC_Grid/Power_Trajectory/rateLimit/Saturation Dynamic'
 * '<S412>' : 'Gen2_ref/HLC_Grid/Subsystem Reference/p2sfilt'
 * '<S413>' : 'Gen2_ref/HLC_Grid/Subsystem Reference/rateLimit1'
 * '<S414>' : 'Gen2_ref/HLC_Grid/Subsystem Reference/p2sfilt/Divisor'
 * '<S415>' : 'Gen2_ref/HLC_Grid/Subsystem Reference/p2sfilt/Divisor/Data Type Conversion Inherited'
 * '<S416>' : 'Gen2_ref/HLC_Grid/Subsystem Reference/rateLimit1/Saturation Dynamic'
 * '<S417>' : 'Gen2_ref/HLC_Island/BDC_Trajectory'
 * '<S418>' : 'Gen2_ref/HLC_Island/CalcPowerRot'
 * '<S419>' : 'Gen2_ref/HLC_Island/DocBlock'
 * '<S420>' : 'Gen2_ref/HLC_Island/Filter'
 * '<S421>' : 'Gen2_ref/HLC_Island/IntegerZOH'
 * '<S422>' : 'Gen2_ref/HLC_Island/LEANOX ERR Correction Transient'
 * '<S423>' : 'Gen2_ref/HLC_Island/LEANOX map'
 * '<S424>' : 'Gen2_ref/HLC_Island/LSL Interface'
 * '<S425>' : 'Gen2_ref/HLC_Island/LVRT freeze'
 * '<S426>' : 'Gen2_ref/HLC_Island/Load Rejection transient compensation'
 * '<S427>' : 'Gen2_ref/HLC_Island/LoadRejection'
 * '<S428>' : 'Gen2_ref/HLC_Island/Model Info'
 * '<S429>' : 'Gen2_ref/HLC_Island/Skip_control'
 * '<S430>' : 'Gen2_ref/HLC_Island/Subsystem'
 * '<S431>' : 'Gen2_ref/HLC_Island/iLQR_SF'
 * '<S432>' : 'Gen2_ref/HLC_Island/p2sFF'
 * '<S433>' : 'Gen2_ref/HLC_Island/BDC_Trajectory/p2sfilt'
 * '<S434>' : 'Gen2_ref/HLC_Island/BDC_Trajectory/rateLimit1'
 * '<S435>' : 'Gen2_ref/HLC_Island/BDC_Trajectory/p2sfilt/Divisor'
 * '<S436>' : 'Gen2_ref/HLC_Island/BDC_Trajectory/p2sfilt/Divisor/Data Type Conversion Inherited'
 * '<S437>' : 'Gen2_ref/HLC_Island/BDC_Trajectory/rateLimit1/Saturation Dynamic'
 * '<S438>' : 'Gen2_ref/HLC_Island/CalcPowerRot/2nd Order Filter'
 * '<S439>' : 'Gen2_ref/HLC_Island/CalcPowerRot/Filter'
 * '<S440>' : 'Gen2_ref/HLC_Island/CalcPowerRot/2nd Order Filter/Divisor1'
 * '<S441>' : 'Gen2_ref/HLC_Island/CalcPowerRot/2nd Order Filter/Divisor1/Data Type Conversion Inherited'
 * '<S442>' : 'Gen2_ref/HLC_Island/CalcPowerRot/Filter/Divisor'
 * '<S443>' : 'Gen2_ref/HLC_Island/CalcPowerRot/Filter/Divisor/Data Type Conversion Inherited'
 * '<S444>' : 'Gen2_ref/HLC_Island/Filter/Divisor'
 * '<S445>' : 'Gen2_ref/HLC_Island/Filter/Divisor/Data Type Conversion Inherited'
 * '<S446>' : 'Gen2_ref/HLC_Island/LEANOX map/Divisor'
 * '<S447>' : 'Gen2_ref/HLC_Island/LEANOX map/Divisor1'
 * '<S448>' : 'Gen2_ref/HLC_Island/LEANOX map/Divisor10'
 * '<S449>' : 'Gen2_ref/HLC_Island/LEANOX map/Divisor11'
 * '<S450>' : 'Gen2_ref/HLC_Island/LEANOX map/Divisor12'
 * '<S451>' : 'Gen2_ref/HLC_Island/LEANOX map/Divisor2'
 * '<S452>' : 'Gen2_ref/HLC_Island/LEANOX map/Divisor3'
 * '<S453>' : 'Gen2_ref/HLC_Island/LEANOX map/Divisor4'
 * '<S454>' : 'Gen2_ref/HLC_Island/LEANOX map/Divisor5'
 * '<S455>' : 'Gen2_ref/HLC_Island/LEANOX map/Divisor6'
 * '<S456>' : 'Gen2_ref/HLC_Island/LEANOX map/Divisor7'
 * '<S457>' : 'Gen2_ref/HLC_Island/LEANOX map/Divisor8'
 * '<S458>' : 'Gen2_ref/HLC_Island/LEANOX map/Divisor9'
 * '<S459>' : 'Gen2_ref/HLC_Island/LEANOX map/LeanoxCorr'
 * '<S460>' : 'Gen2_ref/HLC_Island/LEANOX map/Divisor/Data Type Conversion Inherited'
 * '<S461>' : 'Gen2_ref/HLC_Island/LEANOX map/Divisor1/Data Type Conversion Inherited'
 * '<S462>' : 'Gen2_ref/HLC_Island/LEANOX map/Divisor10/Data Type Conversion Inherited'
 * '<S463>' : 'Gen2_ref/HLC_Island/LEANOX map/Divisor11/Data Type Conversion Inherited'
 * '<S464>' : 'Gen2_ref/HLC_Island/LEANOX map/Divisor12/Data Type Conversion Inherited'
 * '<S465>' : 'Gen2_ref/HLC_Island/LEANOX map/Divisor2/Data Type Conversion Inherited'
 * '<S466>' : 'Gen2_ref/HLC_Island/LEANOX map/Divisor3/Data Type Conversion Inherited'
 * '<S467>' : 'Gen2_ref/HLC_Island/LEANOX map/Divisor4/Data Type Conversion Inherited'
 * '<S468>' : 'Gen2_ref/HLC_Island/LEANOX map/Divisor5/Data Type Conversion Inherited'
 * '<S469>' : 'Gen2_ref/HLC_Island/LEANOX map/Divisor6/Data Type Conversion Inherited'
 * '<S470>' : 'Gen2_ref/HLC_Island/LEANOX map/Divisor7/Data Type Conversion Inherited'
 * '<S471>' : 'Gen2_ref/HLC_Island/LEANOX map/Divisor8/Data Type Conversion Inherited'
 * '<S472>' : 'Gen2_ref/HLC_Island/LEANOX map/Divisor9/Data Type Conversion Inherited'
 * '<S473>' : 'Gen2_ref/HLC_Island/LEANOX map/LeanoxCorr/Leanox_Comp'
 * '<S474>' : 'Gen2_ref/HLC_Island/LEANOX map/LeanoxCorr/Leanox_Comp/2-point interpolation, with extrapolation'
 * '<S475>' : 'Gen2_ref/HLC_Island/LEANOX map/LeanoxCorr/Leanox_Comp/2-point interpolation, with extrapolation1'
 * '<S476>' : 'Gen2_ref/HLC_Island/LEANOX map/LeanoxCorr/Leanox_Comp/Saturation Dynamic'
 * '<S477>' : 'Gen2_ref/HLC_Island/LEANOX map/LeanoxCorr/Leanox_Comp/Saturation Dynamic1'
 * '<S478>' : 'Gen2_ref/HLC_Island/LSL Interface/Filter1'
 * '<S479>' : 'Gen2_ref/HLC_Island/LSL Interface/Saturation Dynamic'
 * '<S480>' : 'Gen2_ref/HLC_Island/LSL Interface/speed Filter'
 * '<S481>' : 'Gen2_ref/HLC_Island/LSL Interface/Filter1/Divisor'
 * '<S482>' : 'Gen2_ref/HLC_Island/LSL Interface/Filter1/Divisor/Data Type Conversion Inherited'
 * '<S483>' : 'Gen2_ref/HLC_Island/LSL Interface/speed Filter/Divisor'
 * '<S484>' : 'Gen2_ref/HLC_Island/LSL Interface/speed Filter/Divisor/Data Type Conversion Inherited'
 * '<S485>' : 'Gen2_ref/HLC_Island/LVRT freeze/Filter'
 * '<S486>' : 'Gen2_ref/HLC_Island/LVRT freeze/TOF'
 * '<S487>' : 'Gen2_ref/HLC_Island/LVRT freeze/Filter/Divisor'
 * '<S488>' : 'Gen2_ref/HLC_Island/LVRT freeze/Filter/Divisor/Data Type Conversion Inherited'
 * '<S489>' : 'Gen2_ref/HLC_Island/LVRT freeze/TOF/Data Type Conversion Inherited'
 * '<S490>' : 'Gen2_ref/HLC_Island/Load Rejection transient compensation/Detect Saturation at LR'
 * '<S491>' : 'Gen2_ref/HLC_Island/Load Rejection transient compensation/Hysterese'
 * '<S492>' : 'Gen2_ref/HLC_Island/Load Rejection transient compensation/TP'
 * '<S493>' : 'Gen2_ref/HLC_Island/Load Rejection transient compensation/TP1'
 * '<S494>' : 'Gen2_ref/HLC_Island/Load Rejection transient compensation/rateLimit'
 * '<S495>' : 'Gen2_ref/HLC_Island/Load Rejection transient compensation/TP/Compare To Zero'
 * '<S496>' : 'Gen2_ref/HLC_Island/Load Rejection transient compensation/TP/Enabled Subsystem'
 * '<S497>' : 'Gen2_ref/HLC_Island/Load Rejection transient compensation/TP/Enabled Subsystem1'
 * '<S498>' : 'Gen2_ref/HLC_Island/Load Rejection transient compensation/TP/Rate Limiter'
 * '<S499>' : 'Gen2_ref/HLC_Island/Load Rejection transient compensation/TP/Rate Limiter/Saturation Dynamic'
 * '<S500>' : 'Gen2_ref/HLC_Island/Load Rejection transient compensation/TP1/Compare To Zero'
 * '<S501>' : 'Gen2_ref/HLC_Island/Load Rejection transient compensation/TP1/Enabled Subsystem'
 * '<S502>' : 'Gen2_ref/HLC_Island/Load Rejection transient compensation/TP1/Enabled Subsystem1'
 * '<S503>' : 'Gen2_ref/HLC_Island/Load Rejection transient compensation/TP1/Rate Limiter'
 * '<S504>' : 'Gen2_ref/HLC_Island/Load Rejection transient compensation/TP1/Rate Limiter/Saturation Dynamic'
 * '<S505>' : 'Gen2_ref/HLC_Island/Load Rejection transient compensation/rateLimit/Saturation Dynamic'
 * '<S506>' : 'Gen2_ref/HLC_Island/LoadRejection/Divisor'
 * '<S507>' : 'Gen2_ref/HLC_Island/LoadRejection/Divisor1'
 * '<S508>' : 'Gen2_ref/HLC_Island/LoadRejection/Divisor2'
 * '<S509>' : 'Gen2_ref/HLC_Island/LoadRejection/Divisor3'
 * '<S510>' : 'Gen2_ref/HLC_Island/LoadRejection/Saturation Dynamic'
 * '<S511>' : 'Gen2_ref/HLC_Island/LoadRejection/TOF'
 * '<S512>' : 'Gen2_ref/HLC_Island/LoadRejection/TOF1'
 * '<S513>' : 'Gen2_ref/HLC_Island/LoadRejection/TOF2'
 * '<S514>' : 'Gen2_ref/HLC_Island/LoadRejection/TOF3'
 * '<S515>' : 'Gen2_ref/HLC_Island/LoadRejection/TP'
 * '<S516>' : 'Gen2_ref/HLC_Island/LoadRejection/TP_ActSat_CBV'
 * '<S517>' : 'Gen2_ref/HLC_Island/LoadRejection/TP_ActSat_TV'
 * '<S518>' : 'Gen2_ref/HLC_Island/LoadRejection/TP_Ign retard'
 * '<S519>' : 'Gen2_ref/HLC_Island/LoadRejection/TP_Misfire_OFF'
 * '<S520>' : 'Gen2_ref/HLC_Island/LoadRejection/TP_Misfire_OFF1'
 * '<S521>' : 'Gen2_ref/HLC_Island/LoadRejection/TP_Misfire_OFF2'
 * '<S522>' : 'Gen2_ref/HLC_Island/LoadRejection/TP_Misfire_ON'
 * '<S523>' : 'Gen2_ref/HLC_Island/LoadRejection/TP_Misfire_ON_2nd time'
 * '<S524>' : 'Gen2_ref/HLC_Island/LoadRejection/rateLimit'
 * '<S525>' : 'Gen2_ref/HLC_Island/LoadRejection/Divisor/Data Type Conversion Inherited'
 * '<S526>' : 'Gen2_ref/HLC_Island/LoadRejection/Divisor1/Data Type Conversion Inherited'
 * '<S527>' : 'Gen2_ref/HLC_Island/LoadRejection/Divisor2/Data Type Conversion Inherited'
 * '<S528>' : 'Gen2_ref/HLC_Island/LoadRejection/Divisor3/Data Type Conversion Inherited'
 * '<S529>' : 'Gen2_ref/HLC_Island/LoadRejection/TOF/Data Type Conversion Inherited'
 * '<S530>' : 'Gen2_ref/HLC_Island/LoadRejection/TOF1/Data Type Conversion Inherited'
 * '<S531>' : 'Gen2_ref/HLC_Island/LoadRejection/TOF2/Data Type Conversion Inherited'
 * '<S532>' : 'Gen2_ref/HLC_Island/LoadRejection/TOF3/Data Type Conversion Inherited'
 * '<S533>' : 'Gen2_ref/HLC_Island/LoadRejection/TP/Compare To Zero'
 * '<S534>' : 'Gen2_ref/HLC_Island/LoadRejection/TP/Enabled Subsystem'
 * '<S535>' : 'Gen2_ref/HLC_Island/LoadRejection/TP/Enabled Subsystem1'
 * '<S536>' : 'Gen2_ref/HLC_Island/LoadRejection/TP/Rate Limiter'
 * '<S537>' : 'Gen2_ref/HLC_Island/LoadRejection/TP/Rate Limiter/Saturation Dynamic'
 * '<S538>' : 'Gen2_ref/HLC_Island/LoadRejection/TP_ActSat_CBV/Compare To Zero'
 * '<S539>' : 'Gen2_ref/HLC_Island/LoadRejection/TP_ActSat_CBV/Enabled Subsystem'
 * '<S540>' : 'Gen2_ref/HLC_Island/LoadRejection/TP_ActSat_CBV/Enabled Subsystem1'
 * '<S541>' : 'Gen2_ref/HLC_Island/LoadRejection/TP_ActSat_CBV/Rate Limiter'
 * '<S542>' : 'Gen2_ref/HLC_Island/LoadRejection/TP_ActSat_CBV/Rate Limiter/Saturation Dynamic'
 * '<S543>' : 'Gen2_ref/HLC_Island/LoadRejection/TP_ActSat_TV/Compare To Zero'
 * '<S544>' : 'Gen2_ref/HLC_Island/LoadRejection/TP_ActSat_TV/Enabled Subsystem'
 * '<S545>' : 'Gen2_ref/HLC_Island/LoadRejection/TP_ActSat_TV/Enabled Subsystem1'
 * '<S546>' : 'Gen2_ref/HLC_Island/LoadRejection/TP_ActSat_TV/Rate Limiter'
 * '<S547>' : 'Gen2_ref/HLC_Island/LoadRejection/TP_ActSat_TV/Rate Limiter/Saturation Dynamic'
 * '<S548>' : 'Gen2_ref/HLC_Island/LoadRejection/TP_Ign retard/Compare To Zero'
 * '<S549>' : 'Gen2_ref/HLC_Island/LoadRejection/TP_Ign retard/Enabled Subsystem'
 * '<S550>' : 'Gen2_ref/HLC_Island/LoadRejection/TP_Ign retard/Enabled Subsystem1'
 * '<S551>' : 'Gen2_ref/HLC_Island/LoadRejection/TP_Ign retard/Rate Limiter'
 * '<S552>' : 'Gen2_ref/HLC_Island/LoadRejection/TP_Ign retard/Rate Limiter/Saturation Dynamic'
 * '<S553>' : 'Gen2_ref/HLC_Island/LoadRejection/TP_Misfire_OFF/Compare To Zero'
 * '<S554>' : 'Gen2_ref/HLC_Island/LoadRejection/TP_Misfire_OFF/Enabled Subsystem'
 * '<S555>' : 'Gen2_ref/HLC_Island/LoadRejection/TP_Misfire_OFF/Enabled Subsystem1'
 * '<S556>' : 'Gen2_ref/HLC_Island/LoadRejection/TP_Misfire_OFF/Rate Limiter'
 * '<S557>' : 'Gen2_ref/HLC_Island/LoadRejection/TP_Misfire_OFF/Rate Limiter/Saturation Dynamic'
 * '<S558>' : 'Gen2_ref/HLC_Island/LoadRejection/TP_Misfire_OFF1/Compare To Zero'
 * '<S559>' : 'Gen2_ref/HLC_Island/LoadRejection/TP_Misfire_OFF1/Enabled Subsystem'
 * '<S560>' : 'Gen2_ref/HLC_Island/LoadRejection/TP_Misfire_OFF1/Enabled Subsystem1'
 * '<S561>' : 'Gen2_ref/HLC_Island/LoadRejection/TP_Misfire_OFF1/Rate Limiter'
 * '<S562>' : 'Gen2_ref/HLC_Island/LoadRejection/TP_Misfire_OFF1/Rate Limiter/Saturation Dynamic'
 * '<S563>' : 'Gen2_ref/HLC_Island/LoadRejection/TP_Misfire_OFF2/Compare To Zero'
 * '<S564>' : 'Gen2_ref/HLC_Island/LoadRejection/TP_Misfire_OFF2/Enabled Subsystem'
 * '<S565>' : 'Gen2_ref/HLC_Island/LoadRejection/TP_Misfire_OFF2/Enabled Subsystem1'
 * '<S566>' : 'Gen2_ref/HLC_Island/LoadRejection/TP_Misfire_OFF2/Rate Limiter'
 * '<S567>' : 'Gen2_ref/HLC_Island/LoadRejection/TP_Misfire_OFF2/Rate Limiter/Saturation Dynamic'
 * '<S568>' : 'Gen2_ref/HLC_Island/LoadRejection/TP_Misfire_ON/Compare To Zero'
 * '<S569>' : 'Gen2_ref/HLC_Island/LoadRejection/TP_Misfire_ON/Enabled Subsystem'
 * '<S570>' : 'Gen2_ref/HLC_Island/LoadRejection/TP_Misfire_ON/Enabled Subsystem1'
 * '<S571>' : 'Gen2_ref/HLC_Island/LoadRejection/TP_Misfire_ON/Rate Limiter'
 * '<S572>' : 'Gen2_ref/HLC_Island/LoadRejection/TP_Misfire_ON/Rate Limiter/Saturation Dynamic'
 * '<S573>' : 'Gen2_ref/HLC_Island/LoadRejection/TP_Misfire_ON_2nd time/Compare To Zero'
 * '<S574>' : 'Gen2_ref/HLC_Island/LoadRejection/TP_Misfire_ON_2nd time/Enabled Subsystem'
 * '<S575>' : 'Gen2_ref/HLC_Island/LoadRejection/TP_Misfire_ON_2nd time/Enabled Subsystem1'
 * '<S576>' : 'Gen2_ref/HLC_Island/LoadRejection/TP_Misfire_ON_2nd time/Rate Limiter'
 * '<S577>' : 'Gen2_ref/HLC_Island/LoadRejection/TP_Misfire_ON_2nd time/Rate Limiter/Saturation Dynamic'
 * '<S578>' : 'Gen2_ref/HLC_Island/LoadRejection/rateLimit/Saturation Dynamic'
 * '<S579>' : 'Gen2_ref/HLC_Island/Skip_control/Filter lam lambda_map_adaption1'
 * '<S580>' : 'Gen2_ref/HLC_Island/Skip_control/Lookup Skipfire'
 * '<S581>' : 'Gen2_ref/HLC_Island/Skip_control/pulsed_skipfire_LR'
 * '<S582>' : 'Gen2_ref/HLC_Island/Skip_control/skipfire_LR_notPulsed'
 * '<S583>' : 'Gen2_ref/HLC_Island/Skip_control/Filter lam lambda_map_adaption1/Divisor'
 * '<S584>' : 'Gen2_ref/HLC_Island/Skip_control/Filter lam lambda_map_adaption1/Divisor/Data Type Conversion Inherited'
 * '<S585>' : 'Gen2_ref/HLC_Island/Skip_control/Lookup Skipfire/Lookup Skipfire Static'
 * '<S586>' : 'Gen2_ref/HLC_Island/Skip_control/Lookup Skipfire/lambda control'
 * '<S587>' : 'Gen2_ref/HLC_Island/Skip_control/Lookup Skipfire/Lookup Skipfire Static/Filter'
 * '<S588>' : 'Gen2_ref/HLC_Island/Skip_control/Lookup Skipfire/Lookup Skipfire Static/Filter1'
 * '<S589>' : 'Gen2_ref/HLC_Island/Skip_control/Lookup Skipfire/Lookup Skipfire Static/Look  up Skipfire'
 * '<S590>' : 'Gen2_ref/HLC_Island/Skip_control/Lookup Skipfire/Lookup Skipfire Static/Saturation Dynamic'
 * '<S591>' : 'Gen2_ref/HLC_Island/Skip_control/Lookup Skipfire/Lookup Skipfire Static/Saturation Dynamic1'
 * '<S592>' : 'Gen2_ref/HLC_Island/Skip_control/Lookup Skipfire/Lookup Skipfire Static/Filter/Divisor'
 * '<S593>' : 'Gen2_ref/HLC_Island/Skip_control/Lookup Skipfire/Lookup Skipfire Static/Filter/Divisor/Data Type Conversion Inherited'
 * '<S594>' : 'Gen2_ref/HLC_Island/Skip_control/Lookup Skipfire/Lookup Skipfire Static/Filter1/Divisor'
 * '<S595>' : 'Gen2_ref/HLC_Island/Skip_control/Lookup Skipfire/Lookup Skipfire Static/Filter1/Divisor/Data Type Conversion Inherited'
 * '<S596>' : 'Gen2_ref/HLC_Island/Skip_control/Lookup Skipfire/Lookup Skipfire Static/Look  up Skipfire/Divisor'
 * '<S597>' : 'Gen2_ref/HLC_Island/Skip_control/Lookup Skipfire/Lookup Skipfire Static/Look  up Skipfire/MATLAB Function'
 * '<S598>' : 'Gen2_ref/HLC_Island/Skip_control/Lookup Skipfire/Lookup Skipfire Static/Look  up Skipfire/Saturation Dynamic'
 * '<S599>' : 'Gen2_ref/HLC_Island/Skip_control/Lookup Skipfire/Lookup Skipfire Static/Look  up Skipfire/Divisor/Data Type Conversion Inherited'
 * '<S600>' : 'Gen2_ref/HLC_Island/Skip_control/Lookup Skipfire/lambda control/Divisor'
 * '<S601>' : 'Gen2_ref/HLC_Island/Skip_control/Lookup Skipfire/lambda control/MATLAB Function'
 * '<S602>' : 'Gen2_ref/HLC_Island/Skip_control/Lookup Skipfire/lambda control/Divisor/Data Type Conversion Inherited'
 * '<S603>' : 'Gen2_ref/HLC_Island/Skip_control/pulsed_skipfire_LR/Detect Increase'
 * '<S604>' : 'Gen2_ref/HLC_Island/Skip_control/pulsed_skipfire_LR/Divisor'
 * '<S605>' : 'Gen2_ref/HLC_Island/Skip_control/pulsed_skipfire_LR/Divisor2'
 * '<S606>' : 'Gen2_ref/HLC_Island/Skip_control/pulsed_skipfire_LR/Hysteresis1'
 * '<S607>' : 'Gen2_ref/HLC_Island/Skip_control/pulsed_skipfire_LR/Saturation Dynamic'
 * '<S608>' : 'Gen2_ref/HLC_Island/Skip_control/pulsed_skipfire_LR/pulsewidth modulation'
 * '<S609>' : 'Gen2_ref/HLC_Island/Skip_control/pulsed_skipfire_LR/Divisor/Data Type Conversion Inherited'
 * '<S610>' : 'Gen2_ref/HLC_Island/Skip_control/pulsed_skipfire_LR/Divisor2/Data Type Conversion Inherited'
 * '<S611>' : 'Gen2_ref/HLC_Island/Skip_control/pulsed_skipfire_LR/pulsewidth modulation/Detect Decrease'
 * '<S612>' : 'Gen2_ref/HLC_Island/Skip_control/pulsed_skipfire_LR/pulsewidth modulation/Divisor'
 * '<S613>' : 'Gen2_ref/HLC_Island/Skip_control/pulsed_skipfire_LR/pulsewidth modulation/SkipPulseWaitTP'
 * '<S614>' : 'Gen2_ref/HLC_Island/Skip_control/pulsed_skipfire_LR/pulsewidth modulation/Divisor/Data Type Conversion Inherited'
 * '<S615>' : 'Gen2_ref/HLC_Island/Skip_control/pulsed_skipfire_LR/pulsewidth modulation/SkipPulseWaitTP/Compare To Zero'
 * '<S616>' : 'Gen2_ref/HLC_Island/Skip_control/pulsed_skipfire_LR/pulsewidth modulation/SkipPulseWaitTP/Enabled Subsystem'
 * '<S617>' : 'Gen2_ref/HLC_Island/Skip_control/pulsed_skipfire_LR/pulsewidth modulation/SkipPulseWaitTP/Enabled Subsystem1'
 * '<S618>' : 'Gen2_ref/HLC_Island/Skip_control/pulsed_skipfire_LR/pulsewidth modulation/SkipPulseWaitTP/Rate Limiter'
 * '<S619>' : 'Gen2_ref/HLC_Island/Skip_control/pulsed_skipfire_LR/pulsewidth modulation/SkipPulseWaitTP/Rate Limiter/Saturation Dynamic'
 * '<S620>' : 'Gen2_ref/HLC_Island/Skip_control/skipfire_LR_notPulsed/MATLAB Function'
 * '<S621>' : 'Gen2_ref/HLC_Island/Skip_control/skipfire_LR_notPulsed/MATLAB Function1'
 * '<S622>' : 'Gen2_ref/HLC_Island/Skip_control/skipfire_LR_notPulsed/Saturation Dynamic2'
 * '<S623>' : 'Gen2_ref/HLC_Island/Skip_control/skipfire_LR_notPulsed/Saturation Dynamic3'
 * '<S624>' : 'Gen2_ref/HLC_Island/Subsystem/Saturation Dynamic1'
 * '<S625>' : 'Gen2_ref/HLC_Island/iLQR_SF/Ke'
 * '<S626>' : 'Gen2_ref/HLC_Island/iLQR_SF/Ke Estimator'
 * '<S627>' : 'Gen2_ref/HLC_Island/iLQR_SF/LQR Controller 3states'
 * '<S628>' : 'Gen2_ref/HLC_Island/iLQR_SF/Lambda Shaping'
 * '<S629>' : 'Gen2_ref/HLC_Island/iLQR_SF/Lookup SkipfireMax'
 * '<S630>' : 'Gen2_ref/HLC_Island/iLQR_SF/Map Adaptation w. Ke Estimate'
 * '<S631>' : 'Gen2_ref/HLC_Island/iLQR_SF/Ref LQR'
 * '<S632>' : 'Gen2_ref/HLC_Island/iLQR_SF/Saturation Dynamic'
 * '<S633>' : 'Gen2_ref/HLC_Island/iLQR_SF/Skipfire'
 * '<S634>' : 'Gen2_ref/HLC_Island/iLQR_SF/delta IT acceptance'
 * '<S635>' : 'Gen2_ref/HLC_Island/iLQR_SF/detect saturation lambda'
 * '<S636>' : 'Gen2_ref/HLC_Island/iLQR_SF/gain scheduling // adaption'
 * '<S637>' : 'Gen2_ref/HLC_Island/iLQR_SF/lambda estimation'
 * '<S638>' : 'Gen2_ref/HLC_Island/iLQR_SF/parameter KF'
 * '<S639>' : 'Gen2_ref/HLC_Island/iLQR_SF/parameter LQR'
 * '<S640>' : 'Gen2_ref/HLC_Island/iLQR_SF/ref traj'
 * '<S641>' : 'Gen2_ref/HLC_Island/iLQR_SF/zero offset tracking'
 * '<S642>' : 'Gen2_ref/HLC_Island/iLQR_SF/Ke/Divisor1'
 * '<S643>' : 'Gen2_ref/HLC_Island/iLQR_SF/Ke/Divisor3'
 * '<S644>' : 'Gen2_ref/HLC_Island/iLQR_SF/Ke/Divisor1/Data Type Conversion Inherited'
 * '<S645>' : 'Gen2_ref/HLC_Island/iLQR_SF/Ke/Divisor3/Data Type Conversion Inherited'
 * '<S646>' : 'Gen2_ref/HLC_Island/iLQR_SF/Ke Estimator/Divisor2'
 * '<S647>' : 'Gen2_ref/HLC_Island/iLQR_SF/Ke Estimator/Divisor3'
 * '<S648>' : 'Gen2_ref/HLC_Island/iLQR_SF/Ke Estimator/Divisor6'
 * '<S649>' : 'Gen2_ref/HLC_Island/iLQR_SF/Ke Estimator/Filter1'
 * '<S650>' : 'Gen2_ref/HLC_Island/iLQR_SF/Ke Estimator/Divisor2/Data Type Conversion Inherited'
 * '<S651>' : 'Gen2_ref/HLC_Island/iLQR_SF/Ke Estimator/Divisor3/Data Type Conversion Inherited'
 * '<S652>' : 'Gen2_ref/HLC_Island/iLQR_SF/Ke Estimator/Divisor6/Data Type Conversion Inherited'
 * '<S653>' : 'Gen2_ref/HLC_Island/iLQR_SF/Ke Estimator/Filter1/Divisor'
 * '<S654>' : 'Gen2_ref/HLC_Island/iLQR_SF/Ke Estimator/Filter1/Divisor/Data Type Conversion Inherited'
 * '<S655>' : 'Gen2_ref/HLC_Island/iLQR_SF/Lambda Shaping/FILTER no delay'
 * '<S656>' : 'Gen2_ref/HLC_Island/iLQR_SF/Lambda Shaping/Filter'
 * '<S657>' : 'Gen2_ref/HLC_Island/iLQR_SF/Lambda Shaping/Saturation Dynamic1'
 * '<S658>' : 'Gen2_ref/HLC_Island/iLQR_SF/Lambda Shaping/Saturation Dynamic2'
 * '<S659>' : 'Gen2_ref/HLC_Island/iLQR_SF/Lambda Shaping/gain scheduling Lambda Proportional control'
 * '<S660>' : 'Gen2_ref/HLC_Island/iLQR_SF/Lambda Shaping/Filter/Divisor'
 * '<S661>' : 'Gen2_ref/HLC_Island/iLQR_SF/Lambda Shaping/Filter/Divisor/Data Type Conversion Inherited'
 * '<S662>' : 'Gen2_ref/HLC_Island/iLQR_SF/Lookup SkipfireMax/Divisor'
 * '<S663>' : 'Gen2_ref/HLC_Island/iLQR_SF/Lookup SkipfireMax/Saturation Dynamic'
 * '<S664>' : 'Gen2_ref/HLC_Island/iLQR_SF/Lookup SkipfireMax/Divisor/Data Type Conversion Inherited'
 * '<S665>' : 'Gen2_ref/HLC_Island/iLQR_SF/Map Adaptation w. Ke Estimate/Filter'
 * '<S666>' : 'Gen2_ref/HLC_Island/iLQR_SF/Map Adaptation w. Ke Estimate/KengMap update'
 * '<S667>' : 'Gen2_ref/HLC_Island/iLQR_SF/Map Adaptation w. Ke Estimate/Subsystem'
 * '<S668>' : 'Gen2_ref/HLC_Island/iLQR_SF/Map Adaptation w. Ke Estimate/Filter/Divisor'
 * '<S669>' : 'Gen2_ref/HLC_Island/iLQR_SF/Map Adaptation w. Ke Estimate/Filter/Divisor/Data Type Conversion Inherited'
 * '<S670>' : 'Gen2_ref/HLC_Island/iLQR_SF/Map Adaptation w. Ke Estimate/KengMap update/Divisor'
 * '<S671>' : 'Gen2_ref/HLC_Island/iLQR_SF/Map Adaptation w. Ke Estimate/KengMap update/Ke Map Update'
 * '<S672>' : 'Gen2_ref/HLC_Island/iLQR_SF/Map Adaptation w. Ke Estimate/KengMap update/MATLAB Function1'
 * '<S673>' : 'Gen2_ref/HLC_Island/iLQR_SF/Map Adaptation w. Ke Estimate/KengMap update/Divisor/Data Type Conversion Inherited'
 * '<S674>' : 'Gen2_ref/HLC_Island/iLQR_SF/Map Adaptation w. Ke Estimate/KengMap update/Ke Map Update/Divisor'
 * '<S675>' : 'Gen2_ref/HLC_Island/iLQR_SF/Map Adaptation w. Ke Estimate/KengMap update/Ke Map Update/Divisor/Data Type Conversion Inherited'
 * '<S676>' : 'Gen2_ref/HLC_Island/iLQR_SF/Map Adaptation w. Ke Estimate/Subsystem/TOF'
 * '<S677>' : 'Gen2_ref/HLC_Island/iLQR_SF/Map Adaptation w. Ke Estimate/Subsystem/TON1'
 * '<S678>' : 'Gen2_ref/HLC_Island/iLQR_SF/Map Adaptation w. Ke Estimate/Subsystem/TP'
 * '<S679>' : 'Gen2_ref/HLC_Island/iLQR_SF/Map Adaptation w. Ke Estimate/Subsystem/TP1'
 * '<S680>' : 'Gen2_ref/HLC_Island/iLQR_SF/Map Adaptation w. Ke Estimate/Subsystem/TOF/Data Type Conversion Inherited'
 * '<S681>' : 'Gen2_ref/HLC_Island/iLQR_SF/Map Adaptation w. Ke Estimate/Subsystem/TON1/Data Type Conversion Inherited'
 * '<S682>' : 'Gen2_ref/HLC_Island/iLQR_SF/Map Adaptation w. Ke Estimate/Subsystem/TP/Compare To Zero'
 * '<S683>' : 'Gen2_ref/HLC_Island/iLQR_SF/Map Adaptation w. Ke Estimate/Subsystem/TP/Enabled Subsystem'
 * '<S684>' : 'Gen2_ref/HLC_Island/iLQR_SF/Map Adaptation w. Ke Estimate/Subsystem/TP/Enabled Subsystem1'
 * '<S685>' : 'Gen2_ref/HLC_Island/iLQR_SF/Map Adaptation w. Ke Estimate/Subsystem/TP/Rate Limiter'
 * '<S686>' : 'Gen2_ref/HLC_Island/iLQR_SF/Map Adaptation w. Ke Estimate/Subsystem/TP/Rate Limiter/Saturation Dynamic'
 * '<S687>' : 'Gen2_ref/HLC_Island/iLQR_SF/Map Adaptation w. Ke Estimate/Subsystem/TP1/Compare To Zero'
 * '<S688>' : 'Gen2_ref/HLC_Island/iLQR_SF/Map Adaptation w. Ke Estimate/Subsystem/TP1/Enabled Subsystem'
 * '<S689>' : 'Gen2_ref/HLC_Island/iLQR_SF/Map Adaptation w. Ke Estimate/Subsystem/TP1/Enabled Subsystem1'
 * '<S690>' : 'Gen2_ref/HLC_Island/iLQR_SF/Map Adaptation w. Ke Estimate/Subsystem/TP1/Rate Limiter'
 * '<S691>' : 'Gen2_ref/HLC_Island/iLQR_SF/Map Adaptation w. Ke Estimate/Subsystem/TP1/Rate Limiter/Saturation Dynamic'
 * '<S692>' : 'Gen2_ref/HLC_Island/iLQR_SF/Ref LQR/Divisor'
 * '<S693>' : 'Gen2_ref/HLC_Island/iLQR_SF/Ref LQR/Divisor1'
 * '<S694>' : 'Gen2_ref/HLC_Island/iLQR_SF/Ref LQR/Divisor2'
 * '<S695>' : 'Gen2_ref/HLC_Island/iLQR_SF/Ref LQR/Saturation Dynamic1'
 * '<S696>' : 'Gen2_ref/HLC_Island/iLQR_SF/Ref LQR/Saturation Dynamic2'
 * '<S697>' : 'Gen2_ref/HLC_Island/iLQR_SF/Ref LQR/Saturation Dynamic3'
 * '<S698>' : 'Gen2_ref/HLC_Island/iLQR_SF/Ref LQR/Saturation Dynamic4'
 * '<S699>' : 'Gen2_ref/HLC_Island/iLQR_SF/Ref LQR/Divisor/Data Type Conversion Inherited'
 * '<S700>' : 'Gen2_ref/HLC_Island/iLQR_SF/Ref LQR/Divisor1/Data Type Conversion Inherited'
 * '<S701>' : 'Gen2_ref/HLC_Island/iLQR_SF/Ref LQR/Divisor2/Data Type Conversion Inherited'
 * '<S702>' : 'Gen2_ref/HLC_Island/iLQR_SF/Skipfire/Filter'
 * '<S703>' : 'Gen2_ref/HLC_Island/iLQR_SF/Skipfire/MATLAB Function'
 * '<S704>' : 'Gen2_ref/HLC_Island/iLQR_SF/Skipfire/Filter/Divisor'
 * '<S705>' : 'Gen2_ref/HLC_Island/iLQR_SF/Skipfire/Filter/Divisor/Data Type Conversion Inherited'
 * '<S706>' : 'Gen2_ref/HLC_Island/iLQR_SF/delta IT acceptance/Delay Retard'
 * '<S707>' : 'Gen2_ref/HLC_Island/iLQR_SF/delta IT acceptance/TON'
 * '<S708>' : 'Gen2_ref/HLC_Island/iLQR_SF/delta IT acceptance/rateLimit'
 * '<S709>' : 'Gen2_ref/HLC_Island/iLQR_SF/delta IT acceptance/Delay Retard/Data Type Conversion Inherited'
 * '<S710>' : 'Gen2_ref/HLC_Island/iLQR_SF/delta IT acceptance/TON/Data Type Conversion Inherited'
 * '<S711>' : 'Gen2_ref/HLC_Island/iLQR_SF/delta IT acceptance/rateLimit/Saturation Dynamic'
 * '<S712>' : 'Gen2_ref/HLC_Island/iLQR_SF/gain scheduling // adaption/Divisor'
 * '<S713>' : 'Gen2_ref/HLC_Island/iLQR_SF/gain scheduling // adaption/Filter'
 * '<S714>' : 'Gen2_ref/HLC_Island/iLQR_SF/gain scheduling // adaption/KengMap update'
 * '<S715>' : 'Gen2_ref/HLC_Island/iLQR_SF/gain scheduling // adaption/KengMap update1'
 * '<S716>' : 'Gen2_ref/HLC_Island/iLQR_SF/gain scheduling // adaption/x_dist1 map update'
 * '<S717>' : 'Gen2_ref/HLC_Island/iLQR_SF/gain scheduling // adaption/Divisor/Data Type Conversion Inherited'
 * '<S718>' : 'Gen2_ref/HLC_Island/iLQR_SF/gain scheduling // adaption/Filter/Divisor'
 * '<S719>' : 'Gen2_ref/HLC_Island/iLQR_SF/gain scheduling // adaption/Filter/Divisor/Data Type Conversion Inherited'
 * '<S720>' : 'Gen2_ref/HLC_Island/iLQR_SF/gain scheduling // adaption/KengMap update/MATLAB Function1'
 * '<S721>' : 'Gen2_ref/HLC_Island/iLQR_SF/gain scheduling // adaption/KengMap update/Saturation Dynamic'
 * '<S722>' : 'Gen2_ref/HLC_Island/iLQR_SF/gain scheduling // adaption/KengMap update/TON'
 * '<S723>' : 'Gen2_ref/HLC_Island/iLQR_SF/gain scheduling // adaption/KengMap update/TON/Data Type Conversion Inherited'
 * '<S724>' : 'Gen2_ref/HLC_Island/iLQR_SF/gain scheduling // adaption/KengMap update1/MATLAB Function1'
 * '<S725>' : 'Gen2_ref/HLC_Island/iLQR_SF/gain scheduling // adaption/KengMap update1/Saturation Dynamic'
 * '<S726>' : 'Gen2_ref/HLC_Island/iLQR_SF/gain scheduling // adaption/KengMap update1/TON'
 * '<S727>' : 'Gen2_ref/HLC_Island/iLQR_SF/gain scheduling // adaption/KengMap update1/TON/Data Type Conversion Inherited'
 * '<S728>' : 'Gen2_ref/HLC_Island/iLQR_SF/gain scheduling // adaption/x_dist1 map update/MATLAB Function'
 * '<S729>' : 'Gen2_ref/HLC_Island/iLQR_SF/gain scheduling // adaption/x_dist1 map update/TON'
 * '<S730>' : 'Gen2_ref/HLC_Island/iLQR_SF/gain scheduling // adaption/x_dist1 map update/TON/Data Type Conversion Inherited'
 * '<S731>' : 'Gen2_ref/HLC_Island/iLQR_SF/lambda estimation/Divisor'
 * '<S732>' : 'Gen2_ref/HLC_Island/iLQR_SF/lambda estimation/Filter'
 * '<S733>' : 'Gen2_ref/HLC_Island/iLQR_SF/lambda estimation/Divisor/Data Type Conversion Inherited'
 * '<S734>' : 'Gen2_ref/HLC_Island/iLQR_SF/lambda estimation/Filter/Divisor'
 * '<S735>' : 'Gen2_ref/HLC_Island/iLQR_SF/lambda estimation/Filter/Divisor/Data Type Conversion Inherited'
 * '<S736>' : 'Gen2_ref/HLC_Island/iLQR_SF/parameter LQR/Divisor'
 * '<S737>' : 'Gen2_ref/HLC_Island/iLQR_SF/parameter LQR/gain scheduling D'
 * '<S738>' : 'Gen2_ref/HLC_Island/iLQR_SF/parameter LQR/gain scheduling LQR'
 * '<S739>' : 'Gen2_ref/HLC_Island/iLQR_SF/parameter LQR/gain scheduling TBDC'
 * '<S740>' : 'Gen2_ref/HLC_Island/iLQR_SF/parameter LQR/gain scheduling T_Lam'
 * '<S741>' : 'Gen2_ref/HLC_Island/iLQR_SF/parameter LQR/Divisor/Data Type Conversion Inherited'
 * '<S742>' : 'Gen2_ref/HLC_Island/iLQR_SF/parameter LQR/gain scheduling D/Divisor'
 * '<S743>' : 'Gen2_ref/HLC_Island/iLQR_SF/parameter LQR/gain scheduling D/Filter'
 * '<S744>' : 'Gen2_ref/HLC_Island/iLQR_SF/parameter LQR/gain scheduling D/Divisor/Data Type Conversion Inherited'
 * '<S745>' : 'Gen2_ref/HLC_Island/iLQR_SF/parameter LQR/gain scheduling D/Filter/Divisor'
 * '<S746>' : 'Gen2_ref/HLC_Island/iLQR_SF/parameter LQR/gain scheduling D/Filter/Divisor/Data Type Conversion Inherited'
 * '<S747>' : 'Gen2_ref/HLC_Island/iLQR_SF/zero offset tracking/Gain Scheduling'
 * '<S748>' : 'Gen2_ref/HLC_Island/iLQR_SF/zero offset tracking/Integration for tracking'
 * '<S749>' : 'Gen2_ref/HLC_Island/iLQR_SF/zero offset tracking/bOutOfNWindow'
 * '<S750>' : 'Gen2_ref/HLC_Island/iLQR_SF/zero offset tracking/Gain Scheduling/TON'
 * '<S751>' : 'Gen2_ref/HLC_Island/iLQR_SF/zero offset tracking/Gain Scheduling/TON/Data Type Conversion Inherited'
 * '<S752>' : 'Gen2_ref/HLC_Island/iLQR_SF/zero offset tracking/Integration for tracking/Anti Wind Up'
 * '<S753>' : 'Gen2_ref/HLC_Island/iLQR_SF/zero offset tracking/Integration for tracking/Anti Wind Up1'
 * '<S754>' : 'Gen2_ref/HLC_Island/iLQR_SF/zero offset tracking/Integration for tracking/Saturation Dynamic'
 * '<S755>' : 'Gen2_ref/HLC_Island/iLQR_SF/zero offset tracking/Integration for tracking/Anti Wind Up/Saturation Dynamic'
 * '<S756>' : 'Gen2_ref/HLC_Island/iLQR_SF/zero offset tracking/Integration for tracking/Anti Wind Up1/Saturation Dynamic1'
 * '<S757>' : 'Gen2_ref/HLC_Island/iLQR_SF/zero offset tracking/bOutOfNWindow/MATLAB Function'
 * '<S758>' : 'Gen2_ref/HLC_Island/p2sFF/LEANOX map'
 * '<S759>' : 'Gen2_ref/HLC_Island/p2sFF/Saturation Dynamic1'
 * '<S760>' : 'Gen2_ref/HLC_Island/p2sFF/Subsystem Reference'
 * '<S761>' : 'Gen2_ref/HLC_Island/p2sFF/Subsystem Reference1'
 * '<S762>' : 'Gen2_ref/HLC_Island/p2sFF/LEANOX map/Divisor'
 * '<S763>' : 'Gen2_ref/HLC_Island/p2sFF/LEANOX map/Divisor1'
 * '<S764>' : 'Gen2_ref/HLC_Island/p2sFF/LEANOX map/Divisor10'
 * '<S765>' : 'Gen2_ref/HLC_Island/p2sFF/LEANOX map/Divisor11'
 * '<S766>' : 'Gen2_ref/HLC_Island/p2sFF/LEANOX map/Divisor12'
 * '<S767>' : 'Gen2_ref/HLC_Island/p2sFF/LEANOX map/Divisor2'
 * '<S768>' : 'Gen2_ref/HLC_Island/p2sFF/LEANOX map/Divisor3'
 * '<S769>' : 'Gen2_ref/HLC_Island/p2sFF/LEANOX map/Divisor4'
 * '<S770>' : 'Gen2_ref/HLC_Island/p2sFF/LEANOX map/Divisor5'
 * '<S771>' : 'Gen2_ref/HLC_Island/p2sFF/LEANOX map/Divisor6'
 * '<S772>' : 'Gen2_ref/HLC_Island/p2sFF/LEANOX map/Divisor7'
 * '<S773>' : 'Gen2_ref/HLC_Island/p2sFF/LEANOX map/Divisor8'
 * '<S774>' : 'Gen2_ref/HLC_Island/p2sFF/LEANOX map/Divisor9'
 * '<S775>' : 'Gen2_ref/HLC_Island/p2sFF/LEANOX map/LeanoxCorr'
 * '<S776>' : 'Gen2_ref/HLC_Island/p2sFF/LEANOX map/Divisor/Data Type Conversion Inherited'
 * '<S777>' : 'Gen2_ref/HLC_Island/p2sFF/LEANOX map/Divisor1/Data Type Conversion Inherited'
 * '<S778>' : 'Gen2_ref/HLC_Island/p2sFF/LEANOX map/Divisor10/Data Type Conversion Inherited'
 * '<S779>' : 'Gen2_ref/HLC_Island/p2sFF/LEANOX map/Divisor11/Data Type Conversion Inherited'
 * '<S780>' : 'Gen2_ref/HLC_Island/p2sFF/LEANOX map/Divisor12/Data Type Conversion Inherited'
 * '<S781>' : 'Gen2_ref/HLC_Island/p2sFF/LEANOX map/Divisor2/Data Type Conversion Inherited'
 * '<S782>' : 'Gen2_ref/HLC_Island/p2sFF/LEANOX map/Divisor3/Data Type Conversion Inherited'
 * '<S783>' : 'Gen2_ref/HLC_Island/p2sFF/LEANOX map/Divisor4/Data Type Conversion Inherited'
 * '<S784>' : 'Gen2_ref/HLC_Island/p2sFF/LEANOX map/Divisor5/Data Type Conversion Inherited'
 * '<S785>' : 'Gen2_ref/HLC_Island/p2sFF/LEANOX map/Divisor6/Data Type Conversion Inherited'
 * '<S786>' : 'Gen2_ref/HLC_Island/p2sFF/LEANOX map/Divisor7/Data Type Conversion Inherited'
 * '<S787>' : 'Gen2_ref/HLC_Island/p2sFF/LEANOX map/Divisor8/Data Type Conversion Inherited'
 * '<S788>' : 'Gen2_ref/HLC_Island/p2sFF/LEANOX map/Divisor9/Data Type Conversion Inherited'
 * '<S789>' : 'Gen2_ref/HLC_Island/p2sFF/LEANOX map/LeanoxCorr/Leanox_Comp'
 * '<S790>' : 'Gen2_ref/HLC_Island/p2sFF/LEANOX map/LeanoxCorr/Leanox_Comp/2-point interpolation, with extrapolation'
 * '<S791>' : 'Gen2_ref/HLC_Island/p2sFF/LEANOX map/LeanoxCorr/Leanox_Comp/2-point interpolation, with extrapolation1'
 * '<S792>' : 'Gen2_ref/HLC_Island/p2sFF/LEANOX map/LeanoxCorr/Leanox_Comp/Saturation Dynamic'
 * '<S793>' : 'Gen2_ref/HLC_Island/p2sFF/LEANOX map/LeanoxCorr/Leanox_Comp/Saturation Dynamic1'
 * '<S794>' : 'Gen2_ref/HLC_Island/p2sFF/Subsystem Reference/p2sfilt'
 * '<S795>' : 'Gen2_ref/HLC_Island/p2sFF/Subsystem Reference/rateLimit1'
 * '<S796>' : 'Gen2_ref/HLC_Island/p2sFF/Subsystem Reference/p2sfilt/Divisor'
 * '<S797>' : 'Gen2_ref/HLC_Island/p2sFF/Subsystem Reference/p2sfilt/Divisor/Data Type Conversion Inherited'
 * '<S798>' : 'Gen2_ref/HLC_Island/p2sFF/Subsystem Reference/rateLimit1/Saturation Dynamic'
 * '<S799>' : 'Gen2_ref/HLC_Island/p2sFF/Subsystem Reference1/Divisor'
 * '<S800>' : 'Gen2_ref/HLC_Island/p2sFF/Subsystem Reference1/Filter'
 * '<S801>' : 'Gen2_ref/HLC_Island/p2sFF/Subsystem Reference1/Filter1'
 * '<S802>' : 'Gen2_ref/HLC_Island/p2sFF/Subsystem Reference1/Divisor/Data Type Conversion Inherited'
 * '<S803>' : 'Gen2_ref/HLC_Island/p2sFF/Subsystem Reference1/Filter/Divisor'
 * '<S804>' : 'Gen2_ref/HLC_Island/p2sFF/Subsystem Reference1/Filter/Divisor/Data Type Conversion Inherited'
 * '<S805>' : 'Gen2_ref/HLC_Island/p2sFF/Subsystem Reference1/Filter1/Divisor'
 * '<S806>' : 'Gen2_ref/HLC_Island/p2sFF/Subsystem Reference1/Filter1/Divisor/Data Type Conversion Inherited'
 * '<S807>' : 'Gen2_ref/ITC/Compare To Constant'
 * '<S808>' : 'Gen2_ref/ITC/DocBlock'
 * '<S809>' : 'Gen2_ref/ITC/Model Info'
 * '<S810>' : 'Gen2_ref/ITC/Saturation Dynamic'
 * '<S811>' : 'Gen2_ref/ITC/rateLimit2'
 * '<S812>' : 'Gen2_ref/ITC/rateLimit2/Saturation Dynamic'
 * '<S813>' : 'Gen2_ref/Ke Estimator NetP/Ke'
 * '<S814>' : 'Gen2_ref/Ke Estimator NetP/Ke Estimator'
 * '<S815>' : 'Gen2_ref/Ke Estimator NetP/Map Adaptation w. Ke Estimate'
 * '<S816>' : 'Gen2_ref/Ke Estimator NetP/Ke/Divisor1'
 * '<S817>' : 'Gen2_ref/Ke Estimator NetP/Ke/Divisor3'
 * '<S818>' : 'Gen2_ref/Ke Estimator NetP/Ke/Divisor1/Data Type Conversion Inherited'
 * '<S819>' : 'Gen2_ref/Ke Estimator NetP/Ke/Divisor3/Data Type Conversion Inherited'
 * '<S820>' : 'Gen2_ref/Ke Estimator NetP/Ke Estimator/Divisor2'
 * '<S821>' : 'Gen2_ref/Ke Estimator NetP/Ke Estimator/Divisor3'
 * '<S822>' : 'Gen2_ref/Ke Estimator NetP/Ke Estimator/Divisor6'
 * '<S823>' : 'Gen2_ref/Ke Estimator NetP/Ke Estimator/Filter1'
 * '<S824>' : 'Gen2_ref/Ke Estimator NetP/Ke Estimator/Divisor2/Data Type Conversion Inherited'
 * '<S825>' : 'Gen2_ref/Ke Estimator NetP/Ke Estimator/Divisor3/Data Type Conversion Inherited'
 * '<S826>' : 'Gen2_ref/Ke Estimator NetP/Ke Estimator/Divisor6/Data Type Conversion Inherited'
 * '<S827>' : 'Gen2_ref/Ke Estimator NetP/Ke Estimator/Filter1/Divisor'
 * '<S828>' : 'Gen2_ref/Ke Estimator NetP/Ke Estimator/Filter1/Divisor/Data Type Conversion Inherited'
 * '<S829>' : 'Gen2_ref/Ke Estimator NetP/Map Adaptation w. Ke Estimate/Filter'
 * '<S830>' : 'Gen2_ref/Ke Estimator NetP/Map Adaptation w. Ke Estimate/KengMap update'
 * '<S831>' : 'Gen2_ref/Ke Estimator NetP/Map Adaptation w. Ke Estimate/Subsystem'
 * '<S832>' : 'Gen2_ref/Ke Estimator NetP/Map Adaptation w. Ke Estimate/Filter/Divisor'
 * '<S833>' : 'Gen2_ref/Ke Estimator NetP/Map Adaptation w. Ke Estimate/Filter/Divisor/Data Type Conversion Inherited'
 * '<S834>' : 'Gen2_ref/Ke Estimator NetP/Map Adaptation w. Ke Estimate/KengMap update/Divisor'
 * '<S835>' : 'Gen2_ref/Ke Estimator NetP/Map Adaptation w. Ke Estimate/KengMap update/Ke Map Update'
 * '<S836>' : 'Gen2_ref/Ke Estimator NetP/Map Adaptation w. Ke Estimate/KengMap update/MATLAB Function1'
 * '<S837>' : 'Gen2_ref/Ke Estimator NetP/Map Adaptation w. Ke Estimate/KengMap update/Divisor/Data Type Conversion Inherited'
 * '<S838>' : 'Gen2_ref/Ke Estimator NetP/Map Adaptation w. Ke Estimate/KengMap update/Ke Map Update/Divisor'
 * '<S839>' : 'Gen2_ref/Ke Estimator NetP/Map Adaptation w. Ke Estimate/KengMap update/Ke Map Update/Divisor/Data Type Conversion Inherited'
 * '<S840>' : 'Gen2_ref/Ke Estimator NetP/Map Adaptation w. Ke Estimate/Subsystem/TOF'
 * '<S841>' : 'Gen2_ref/Ke Estimator NetP/Map Adaptation w. Ke Estimate/Subsystem/TON1'
 * '<S842>' : 'Gen2_ref/Ke Estimator NetP/Map Adaptation w. Ke Estimate/Subsystem/TP'
 * '<S843>' : 'Gen2_ref/Ke Estimator NetP/Map Adaptation w. Ke Estimate/Subsystem/TP1'
 * '<S844>' : 'Gen2_ref/Ke Estimator NetP/Map Adaptation w. Ke Estimate/Subsystem/TOF/Data Type Conversion Inherited'
 * '<S845>' : 'Gen2_ref/Ke Estimator NetP/Map Adaptation w. Ke Estimate/Subsystem/TON1/Data Type Conversion Inherited'
 * '<S846>' : 'Gen2_ref/Ke Estimator NetP/Map Adaptation w. Ke Estimate/Subsystem/TP/Compare To Zero'
 * '<S847>' : 'Gen2_ref/Ke Estimator NetP/Map Adaptation w. Ke Estimate/Subsystem/TP/Enabled Subsystem'
 * '<S848>' : 'Gen2_ref/Ke Estimator NetP/Map Adaptation w. Ke Estimate/Subsystem/TP/Enabled Subsystem1'
 * '<S849>' : 'Gen2_ref/Ke Estimator NetP/Map Adaptation w. Ke Estimate/Subsystem/TP/Rate Limiter'
 * '<S850>' : 'Gen2_ref/Ke Estimator NetP/Map Adaptation w. Ke Estimate/Subsystem/TP/Rate Limiter/Saturation Dynamic'
 * '<S851>' : 'Gen2_ref/Ke Estimator NetP/Map Adaptation w. Ke Estimate/Subsystem/TP1/Compare To Zero'
 * '<S852>' : 'Gen2_ref/Ke Estimator NetP/Map Adaptation w. Ke Estimate/Subsystem/TP1/Enabled Subsystem'
 * '<S853>' : 'Gen2_ref/Ke Estimator NetP/Map Adaptation w. Ke Estimate/Subsystem/TP1/Enabled Subsystem1'
 * '<S854>' : 'Gen2_ref/Ke Estimator NetP/Map Adaptation w. Ke Estimate/Subsystem/TP1/Rate Limiter'
 * '<S855>' : 'Gen2_ref/Ke Estimator NetP/Map Adaptation w. Ke Estimate/Subsystem/TP1/Rate Limiter/Saturation Dynamic'
 * '<S856>' : 'Gen2_ref/LHV estimator/Divisor'
 * '<S857>' : 'Gen2_ref/LHV estimator/Divisor/Data Type Conversion Inherited'
 * '<S858>' : 'Gen2_ref/LambdaLimit/Divisor'
 * '<S859>' : 'Gen2_ref/LambdaLimit/Filter'
 * '<S860>' : 'Gen2_ref/LambdaLimit/Saturation Dynamic'
 * '<S861>' : 'Gen2_ref/LambdaLimit/Saturation Dynamic1'
 * '<S862>' : 'Gen2_ref/LambdaLimit/Divisor/Data Type Conversion Inherited'
 * '<S863>' : 'Gen2_ref/LambdaLimit/Filter/Divisor'
 * '<S864>' : 'Gen2_ref/LambdaLimit/Filter/Divisor/Data Type Conversion Inherited'
 * '<S865>' : 'Gen2_ref/Leanox_Comp_WG/CD_map'
 * '<S866>' : 'Gen2_ref/Leanox_Comp_WG/Filter1'
 * '<S867>' : 'Gen2_ref/Leanox_Comp_WG/LookUp Extrapolation'
 * '<S868>' : 'Gen2_ref/Leanox_Comp_WG/ThetaCD_aux'
 * '<S869>' : 'Gen2_ref/Leanox_Comp_WG/Filter1/Divisor'
 * '<S870>' : 'Gen2_ref/Leanox_Comp_WG/Filter1/Divisor/Data Type Conversion Inherited'
 * '<S871>' : 'Gen2_ref/Leanox_Comp_WG/ThetaCD_aux/Divisor'
 * '<S872>' : 'Gen2_ref/Leanox_Comp_WG/ThetaCD_aux/Divisor/Data Type Conversion Inherited'
 * '<S873>' : 'Gen2_ref/Outputs/FILTER no delay'
 * '<S874>' : 'Gen2_ref/Power trajectory/LVRT_React'
 * '<S875>' : 'Gen2_ref/Power trajectory/Power_Trajectory'
 * '<S876>' : 'Gen2_ref/Power trajectory/LVRT_React/MATLAB Function'
 * '<S877>' : 'Gen2_ref/Power trajectory/Power_Trajectory/Pd_filt'
 * '<S878>' : 'Gen2_ref/Power trajectory/Power_Trajectory/Saturation Dynamic'
 * '<S879>' : 'Gen2_ref/Power trajectory/Power_Trajectory/Saturation Dynamic1'
 * '<S880>' : 'Gen2_ref/Power trajectory/Power_Trajectory/Saturation Dynamic2'
 * '<S881>' : 'Gen2_ref/Power trajectory/Power_Trajectory/rateLimit'
 * '<S882>' : 'Gen2_ref/Power trajectory/Power_Trajectory/Pd_filt/Divisor'
 * '<S883>' : 'Gen2_ref/Power trajectory/Power_Trajectory/Pd_filt/Divisor/Data Type Conversion Inherited'
 * '<S884>' : 'Gen2_ref/Power trajectory/Power_Trajectory/rateLimit/Saturation Dynamic'
 * '<S885>' : 'Gen2_ref/Skipfire/DocBlock'
 * '<S886>' : 'Gen2_ref/Skipfire/Filter'
 * '<S887>' : 'Gen2_ref/Skipfire/Filter1'
 * '<S888>' : 'Gen2_ref/Skipfire/Lookup Skipfire'
 * '<S889>' : 'Gen2_ref/Skipfire/Lookup SkipfireMax'
 * '<S890>' : 'Gen2_ref/Skipfire/MATLAB Function'
 * '<S891>' : 'Gen2_ref/Skipfire/Model Info'
 * '<S892>' : 'Gen2_ref/Skipfire/Saturation Dynamic'
 * '<S893>' : 'Gen2_ref/Skipfire/Saturation Dynamic1'
 * '<S894>' : 'Gen2_ref/Skipfire/Saturation Dynamic2'
 * '<S895>' : 'Gen2_ref/Skipfire/Saturation Dynamic3'
 * '<S896>' : 'Gen2_ref/Skipfire/Skip_control_type3_4'
 * '<S897>' : 'Gen2_ref/Skipfire/Filter/Divisor'
 * '<S898>' : 'Gen2_ref/Skipfire/Filter/Divisor/Data Type Conversion Inherited'
 * '<S899>' : 'Gen2_ref/Skipfire/Filter1/Divisor'
 * '<S900>' : 'Gen2_ref/Skipfire/Filter1/Divisor/Data Type Conversion Inherited'
 * '<S901>' : 'Gen2_ref/Skipfire/Lookup Skipfire/Divisor'
 * '<S902>' : 'Gen2_ref/Skipfire/Lookup Skipfire/Saturation Dynamic'
 * '<S903>' : 'Gen2_ref/Skipfire/Lookup Skipfire/Divisor/Data Type Conversion Inherited'
 * '<S904>' : 'Gen2_ref/Skipfire/Lookup SkipfireMax/Divisor'
 * '<S905>' : 'Gen2_ref/Skipfire/Lookup SkipfireMax/Saturation Dynamic'
 * '<S906>' : 'Gen2_ref/Skipfire/Lookup SkipfireMax/Divisor/Data Type Conversion Inherited'
 * '<S907>' : 'Gen2_ref/Skipfire/Skip_control_type3_4/Saturation Dynamic2'
 * '<S908>' : 'Gen2_ref/SteadyState/Divisor'
 * '<S909>' : 'Gen2_ref/SteadyState/Enabled Subsystem2'
 * '<S910>' : 'Gen2_ref/SteadyState/Filter'
 * '<S911>' : 'Gen2_ref/SteadyState/Filter1'
 * '<S912>' : 'Gen2_ref/SteadyState/Filter2'
 * '<S913>' : 'Gen2_ref/SteadyState/Filter3'
 * '<S914>' : 'Gen2_ref/SteadyState/TON'
 * '<S915>' : 'Gen2_ref/SteadyState/TON1'
 * '<S916>' : 'Gen2_ref/SteadyState/TON2'
 * '<S917>' : 'Gen2_ref/SteadyState/timer'
 * '<S918>' : 'Gen2_ref/SteadyState/Divisor/Data Type Conversion Inherited'
 * '<S919>' : 'Gen2_ref/SteadyState/Filter/Divisor'
 * '<S920>' : 'Gen2_ref/SteadyState/Filter/Divisor/Data Type Conversion Inherited'
 * '<S921>' : 'Gen2_ref/SteadyState/Filter1/Divisor'
 * '<S922>' : 'Gen2_ref/SteadyState/Filter1/Divisor/Data Type Conversion Inherited'
 * '<S923>' : 'Gen2_ref/SteadyState/Filter2/Divisor'
 * '<S924>' : 'Gen2_ref/SteadyState/Filter2/Divisor/Data Type Conversion Inherited'
 * '<S925>' : 'Gen2_ref/SteadyState/Filter3/Divisor'
 * '<S926>' : 'Gen2_ref/SteadyState/Filter3/Divisor/Data Type Conversion Inherited'
 * '<S927>' : 'Gen2_ref/SteadyState/TON/Data Type Conversion Inherited'
 * '<S928>' : 'Gen2_ref/SteadyState/TON1/Data Type Conversion Inherited'
 * '<S929>' : 'Gen2_ref/SteadyState/TON2/Data Type Conversion Inherited'
 */
#endif                                 /* RTW_HEADER_Gen2_ref_h_ */
```

#### Gen2_ref_data.c
```c
/********************************************************************
 * COPYRIGHT -- B&R Industrial Automation GmbH
 ********************************************************************
 * Program: Gen2_ref
 * File: Gen2_ref_data.c
 * Author: 105055527
 * Last modified by: kelleto00
 * Created: Wed Apr 16 13:02:53 2008
 * Last modified: Wed Oct 09 10:01:33 2024
 * Model Version: 4.14.00.04
 * Description: V4.10.00.01, 01-09-2020 Keller, Ke Estimator, additive LS factor, Ptraj SpeedCtrl, LVRT Freeze HLCi
   V4.10.00.01, 02-10-2020 Keller, bugfix HLCi p2srefLX init, BDC_lib: change Inf to 1e7
   V4.10.00.01, 13-11-2020 Keller, bugfix LXcorr T2s/ZZP, LSLff damping, dbgOut for Leanox WG compensation
   V4.10.00.01, 27-01-2021 Keller, Lx WGV compensation: no reset in island mode, addition before skipfire compensation
   V4.10.00.01, 02-02-2021 Keller, initialization lambda estimation with rLam_Start
   V4.11.00.01, 28-05-2021 Keller, Gas Quality Change (GQC) Improvements, LHV estimator output
   V4.11.00.01, 05-11-2021 Keller, Bugfix BDC: worksplit offset, optionally Nset instead of Nnom, rN_Eng_LRskipF
   V4.12.00.01, 10-02-2021 Keller, SpeedCtrl2.0 TU Wien: Disturbance Estimator, LQR incl. droop & leanox
   V4.12.00.02, 23-05-2022 Arnold, Leanox point C in low load
   V4.12.00.02, 09-06-2022 Kafka, add external skip fire input for isolated and grid parallel operation
   V4.12.00.03, 15-09-2022 Keller, add power trajectory to HLCi for extended LQR (Droop setpoint)
   V4.12.00.04, 12-10-2022 Keller, add gas flow comp. factor for rejections
   V4.12.00.05, 13-10-2022 Keller, power filter for static skipfire in island mode
   V4.12.00.06, 15-11-2022 Keller, Ke adaptation with disturbance observer
   V4.13.00.01, 15-11-2022 Keller, FDC: R_mix output, HLCi: R_mix for Ke
   V4.13.00.02, 10-07-2023 Keller, interpolation of LHV, rho_gas and Lmin
   V4.13.00.03, 10-07-2023 Keller, load dependent gas dosage delay
   V4.13.00.04, 11-09-2023 Keller, D-part FSM, bugfix dPTV ramp
   V4.13.00.05, 27-02-2024 Keller, Filter outputs without bSS
   V4.13.00.06, 10-04-2024 Keller, bugfix leanox manual mode with bSepEmisCtrl
   V4.14.00.01, 01-07-2024 Keller, iNskip_LRfor Ke calculation
   V4.14.00.02, 17-09-2024 Keller, Use actual speed for observer disturbance dg (Gen2_ref/HLC_Island (HLC_Island_ref)/iLQR_SF/Ref LQR)
   V4.14.00.03, 30-09-2024 Keller, LR gas flow compensation possible without actuator saturation
   V4.14.00.04, 02-10-2024 Keller, Limit derivative power setpoint for FSM
 * modified Comment:
 ********************************************************************
 * Data for program Gen2_ref
 ********************************************************************
 * Generated with B&R Automation Studio Target for Simulink V6.7.1
 * (ERT based)
 ********************************************************************/

#include "Gen2_ref.h"
#include "Gen2_ref_private.h"

/*  GLOBAL DATA DEFINITIONS */

/* Invariant block signals (default storage) */
const ConstBlockIO_Gen2_ref Gen2_ref_ConstB = {
  0.0,                                 /* '<S62>/Constant11' */
  1.0,                                 /* '<S134>/  1' */
  0.0,                                 /* '<S344>/ tde1' */
  0.0,                                 /* '<S628>/Constant2' */
  0.0,                                 /* '<S633>/Constant3' */
  0.0,                                 /* '<S761>/Constant1' */
  0.0,                                 /* '<S19>/  x0' */
  1.0,                                 /* '<S20>/T_filt1' */

  /* Start of '<S830>/Ke Map Update' */
  {
    0.0                                /* '<S835>/Constant1' */
  }
  ,

  /* End of '<S830>/Ke Map Update' */

  /* Start of '<S636>/Filter' */
  {
    10.0,                              /* '<S718>/Abs' */
    10.0,                              /* '<S718>/Switch' */
    0,                                 /* '<S718>/Relational Operator' */
    1,                                 /* '<S713>/Relational Operator' */
    0                                  /* '<S713>/Logical Operator1' */
  }
  ,

  /* End of '<S636>/Filter' */

  /* Start of '<S666>/Ke Map Update' */
  {
    0.0                                /* '<S671>/Constant1' */
  }
  ,

  /* End of '<S666>/Ke Map Update' */

  /* Start of '<S630>/Filter' */
  {
    10.0,                              /* '<S668>/Abs' */
    10.0,                              /* '<S668>/Switch' */
    0,                                 /* '<S668>/Relational Operator' */
    1,                                 /* '<S665>/Relational Operator' */
    0                                  /* '<S665>/Logical Operator1' */
  }
  ,

  /* End of '<S630>/Filter' */

  /* Start of '<S418>/2nd Order Filter' */
  {
    0.0                                /* '<S438>/Constant' */
  }
  ,

  /* End of '<S418>/2nd Order Filter' */

  /* Start of '<S306>/2nd Order Filter3' */
  {
    0.0                                /* '<S317>/Constant' */
  }
  ,

  /* End of '<S306>/2nd Order Filter3' */

  /* Start of '<S306>/2nd Order Filter2' */
  {
    0.0                                /* '<S316>/Constant' */
  }
  ,

  /* End of '<S306>/2nd Order Filter2' */

  /* Start of '<S306>/2nd Order Filter1' */
  {
    0.0                                /* '<S315>/Constant' */
  }
  ,

  /* End of '<S306>/2nd Order Filter1' */

  /* Start of '<S306>/2nd Order Filter' */
  {
    0.0                                /* '<S314>/Constant' */
  }
  /* End of '<S306>/2nd Order Filter' */
};

/* Constant parameters (default storage) */
const ConstParam_Gen2_ref Gen2_ref_ConstP = {
  /* Expression: [0 0 70 70]
   * Referenced by: '<S134>/LT%2deg'
   */
  { 0.0, 0.0, 70.0, 70.0 },

  /* Expression: [0 0.0625 0.9375 1]
   * Referenced by: '<S134>/LT%2deg'
   */
  { 0.0, 0.0625, 0.9375, 1.0 }
};
```
